RoboDK station: Config_2_New_Drillbit.rdk

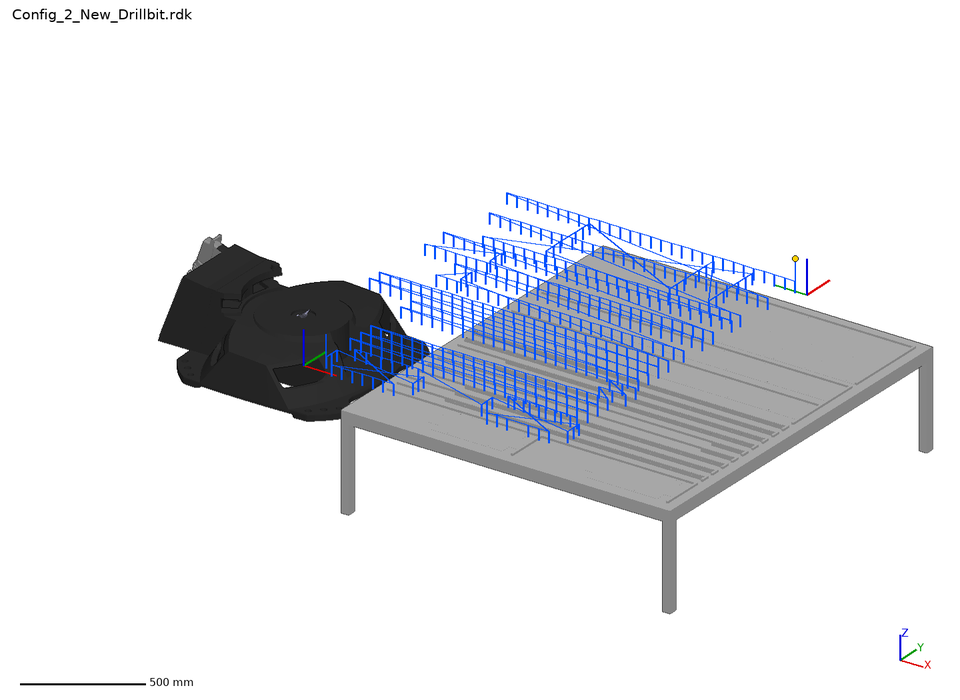
[picture v0: the station drawn from its stored meshes, robots at their saved joint values, targets as dots, program paths as lines]
Station Config_2_New_Drillbit (saved by RoboDK 5.2.3). Poses are relative to the parent item; angles as X-Y-Z fixed-axis rotations.
  - frame KUKA KR 210 R2700 extra Base at (0, 0, 0) mm
    - robot KUKA KR 210 R2700 extra: 6 axes, payload 210 kg, reach 2696 mm, repeatability 0.06 mm, weight 1068 kg
        joint limits [-185, -140, -120, -350, -125, -350] to [185, -5, 155, 350, 125, 350]; home [0, -90, 90, 0, 0, 0]; saved at [43.452, -82.309, 119.903, -52.09, 33.269, 83.396]
      - tool Spindle, TCP at (32, 0, 260) mm, rotated rx 0 ry 39 rz 0 deg, size 157.3 x 72 x 259.9 mm
  - frame Corner First Plate at (1872.67, 817.07, 510.8) mm, rotated rx 0 ry 0 rz 90 deg
  - object Table 2 at (1700, -800, 455) mm, rotated rx 0 ry 0 rz 90 deg, size 1820 x 1600 x 475 mm, geometry from Table 2.stl
  - machining project Path1 settings: rotZ(0) | rotX(0)*rotY(0) | rotz(0) | onStart | onPathStart | onApproach | onPoint | onRetract | onFinish | SetRPM(%1) | SetTool(%1) | Extruder(%1) | default | default | OutOnMov(%1) | OutOffMov(%1) | onPathFinish | M_RunCode(%1)
  - program Path1 (1332 instructions, listed below)
  - object Config_2 at (2494.97, 660, 510.8) mm, rotated rx 0 ry 0 rz 90 deg
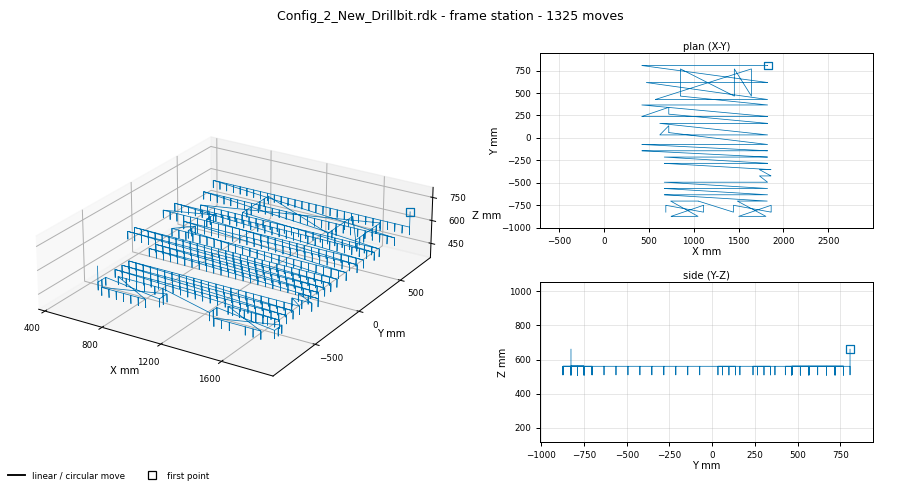
[picture p0: tool path of Config_2_New_Drillbit.rdk in frame station, 1325 of 1325 moves have a stored position in this frame; points joined in program order, loops and branches not executed]

--- program Path1 (robot KUKA KR 210 R2700 extra) ---
  Smooth(1)
  Set speed (1000.0 mm/s)
  Set Ref.: Corner First Plate
  Set Tool: Spindle
  Show Spindle
  MoveJ 1 to (-10.8, 50, 150) mm, rotated rx 180 ry 0 rz 90 deg; joints [-16.649, -45.764, 65.76, 18.984, 33.661, -29.061]
  MoveL 2 to (-10.8, 50, 150) mm, rotated rx 180 ry 0 rz 90 deg; joints [-16.649, -45.764, 65.76, 18.984, 33.661, -29.061]
  MoveL 3 to (-10.8, 50, 50) mm, rotated rx -180 ry 0 rz 90 deg; joints [-16.649, -43.606, 67.21, 20.96, 30.269, -31.389]
  MoveL 4 to (-10.8, 50, 50) mm, rotated rx -180 ry 0 rz 90 deg; joints [-16.649, -43.606, 67.21, 20.96, 30.269, -31.389]
  Set speed (150.0 mm/s)
  MoveL 5 to (-10.8, 50, -0.5) mm, rotated rx -180 ry 0 rz 90 deg; joints [-16.649, -42.409, 67.769, 22.101, 28.635, -32.7]
  MoveL 6 to (-10.8, 50, 50) mm, rotated rx -180 ry 0 rz 90 deg; joints [-16.649, -43.606, 67.21, 20.96, 30.269, -31.389]
  MoveL 7 to (-10.8, 100, 50) mm, rotated rx -180 ry 0 rz 90 deg; joints [-17.019, -45.862, 71.181, 22.479, 28.8, -33.311]
  MoveL 8 to (-10.8, 100, -0.5) mm, rotated rx 180 ry 0 rz 90 deg; joints [-17.019, -44.623, 71.727, 23.8, 27.158, -34.807]
  MoveL 9 to (-10.8, 100, 50) mm, rotated rx -180 ry 0 rz 90 deg; joints [-17.019, -45.862, 71.181, 22.479, 28.8, -33.311]
  MoveL 10 to (-10.8, 150, 50) mm, rotated rx -180 ry 0 rz 90 deg; joints [-17.405, -48.036, 74.965, 24.096, 27.458, -35.338]
  MoveL 11 to (-10.8, 150, -0.5) mm, rotated rx 180 ry 0 rz 90 deg; joints [-17.405, -46.754, 75.501, 25.621, 25.807, -37.043]
  MoveL 12 to (-10.8, 150, 50) mm, rotated rx -180 ry 0 rz 90 deg; joints [-17.405, -48.036, 74.965, 24.096, 27.458, -35.338]
  MoveL 13 to (-10.8, 200, 50) mm, rotated rx 180 ry 0 rz 90 deg; joints [-17.809, -50.14, 78.588, 25.815, 26.232, -37.474]
  MoveL 14 to (-10.8, 200, -0.5) mm, rotated rx 180 ry 0 rz 90 deg; joints [-17.809, -48.815, 79.118, 27.57, 24.574, -39.418]
  MoveL 15 to (-10.8, 200, 50) mm, rotated rx 180 ry 0 rz 90 deg; joints [-17.809, -50.14, 78.588, 25.815, 26.232, -37.474]
  MoveL 16 to (-10.8, 250, 50) mm, rotated rx -180 ry 0 rz 90 deg; joints [-18.231, -52.187, 82.07, 27.638, 25.115, -39.725]
  MoveL 17 to (-10.8, 250, -0.5) mm, rotated rx 180 ry 0 rz 90 deg; joints [-18.231, -50.817, 82.596, 29.652, 23.451, -41.935]
  MoveL 18 to (-10.8, 250, 50) mm, rotated rx -180 ry 0 rz 90 deg; joints [-18.231, -52.187, 82.07, 27.638, 25.115, -39.725]
  MoveL 19 to (-10.8, 300, 50) mm, rotated rx 180 ry 0 rz 90 deg; joints [-18.673, -54.185, 85.428, 29.564, 24.103, -42.091]
  MoveL 20 to (-10.8, 300, -0.5) mm, rotated rx 180 ry 0 rz 90 deg; joints [-18.673, -52.771, 85.952, 31.867, 22.436, -44.597]
  MoveL 21 to (-10.8, 300, 50) mm, rotated rx 180 ry 0 rz 90 deg; joints [-18.673, -54.185, 85.428, 29.564, 24.103, -42.091]
  MoveL 22 to (-10.8, 350, 50) mm, rotated rx -180 ry 0 rz 90 deg; joints [-19.137, -56.143, 88.676, 31.591, 23.192, -44.571]
  MoveL 23 to (-10.8, 350, -0.5) mm, rotated rx 180 ry 0 rz 90 deg; joints [-19.137, -54.682, 89.199, 34.212, 21.526, -47.404]
  MoveL 24 to (-10.8, 350, 50) mm, rotated rx -180 ry 0 rz 90 deg; joints [-19.137, -56.143, 88.676, 31.591, 23.192, -44.571]
  MoveL 25 to (-10.8, 400, 50) mm, rotated rx -180 ry 0 rz 90 deg; joints [-19.622, -58.067, 91.823, 33.712, 22.382, -47.16]
  MoveL 26 to (-10.8, 400, -0.5) mm, rotated rx -180 ry 0 rz 90 deg; joints [-19.622, -56.558, 92.348, 36.68, 20.72, -50.35]
  MoveL 27 to (-10.8, 400, 50) mm, rotated rx -180 ry 0 rz 90 deg; joints [-19.622, -58.067, 91.823, 33.712, 22.382, -47.16]
  MoveL 28 to (-10.8, 450, 50) mm, rotated rx -180 ry 0 rz 90 deg; joints [-20.133, -59.963, 94.88, 35.917, 21.67, -49.848]
  MoveL 29 to (-10.8, 450, -0.5) mm, rotated rx -180 ry 0 rz 90 deg; joints [-20.133, -58.405, 95.407, 39.259, 20.016, -53.424]
  MoveL 30 to (-10.8, 450, 50) mm, rotated rx -180 ry 0 rz 90 deg; joints [-20.133, -59.963, 94.88, 35.917, 21.67, -49.848]
  MoveL 31 to (-10.8, 500, 50) mm, rotated rx 180 ry 0 rz 90 deg; joints [-20.669, -61.837, 97.853, 38.19, 21.055, -52.623]
  MoveL 32 to (-10.8, 500, -0.5) mm, rotated rx -180 ry 0 rz 90 deg; joints [-20.669, -60.228, 98.385, 41.93, 19.415, -56.608]
  MoveL 33 to (-10.8, 500, 50) mm, rotated rx 180 ry 0 rz 90 deg; joints [-20.669, -61.837, 97.853, 38.19, 21.055, -52.623]
  MoveL 34 to (-10.8, 550, 50) mm, rotated rx 180 ry 0 rz 90 deg; joints [-21.233, -63.694, 100.75, 40.513, 20.539, -55.467]
  MoveL 35 to (-10.8, 550, -0.5) mm, rotated rx 180 ry 0 rz 90 deg; joints [-21.233, -62.031, 101.287, 44.668, 18.917, -59.88]
  MoveL 36 to (-10.8, 550, 50) mm, rotated rx 180 ry 0 rz 90 deg; joints [-21.233, -63.694, 100.75, 40.513, 20.539, -55.467]
  MoveL 37 to (-10.8, 600, 50) mm, rotated rx -180 ry 0 rz 90 deg; joints [-21.827, -65.538, 103.574, 42.862, 20.119, -58.358]
  MoveL 38 to (-10.8, 600, -0.5) mm, rotated rx -180 ry 0 rz 90 deg; joints [-21.827, -63.818, 104.119, 47.443, 18.521, -63.211]
  MoveL 39 to (-10.8, 600, 50) mm, rotated rx -180 ry 0 rz 90 deg; joints [-21.827, -65.538, 103.574, 42.862, 20.119, -58.358]
  MoveL 40 to (-10.8, 650, 50) mm, rotated rx 180 ry 0 rz 90 deg; joints [-22.454, -67.373, 106.332, 45.21, 19.797, -61.271]
  MoveL 41 to (-10.8, 650, -0.5) mm, rotated rx 180 ry 0 rz 90 deg; joints [-22.454, -65.594, 106.885, 50.217, 18.226, -66.566]
  MoveL 42 to (-10.8, 650, 50) mm, rotated rx 180 ry 0 rz 90 deg; joints [-22.454, -67.373, 106.332, 45.21, 19.797, -61.271]
  MoveL 43 to (-10.8, 700, 50) mm, rotated rx 180 ry 0 rz 90 deg; joints [-23.115, -69.204, 109.027, 47.525, 19.57, -64.175]
  MoveL 44 to (-10.8, 700, -0.5) mm, rotated rx 180 ry 0 rz 90 deg; joints [-23.115, -67.363, 109.589, 52.952, 18.032, -69.908]
  MoveL 45 to (-10.8, 700, 50) mm, rotated rx 180 ry 0 rz 90 deg; joints [-23.115, -69.204, 109.027, 47.525, 19.57, -64.175]
  MoveL 46 to (-10.8, 750, 50) mm, rotated rx 180 ry 0 rz 90 deg; joints [-23.815, -71.034, 111.662, 49.774, 19.44, -67.041]
  MoveL 47 to (-10.8, 750, -0.5) mm, rotated rx -180 ry 0 rz 90 deg; joints [-23.815, -69.128, 112.235, 55.606, 17.935, -73.196]
  MoveL 48 to (-10.8, 750, 50) mm, rotated rx 180 ry 0 rz 90 deg; joints [-23.815, -71.034, 111.662, 49.774, 19.44, -67.041]
  MoveL 49 to (-10.8, 800, 50) mm, rotated rx -180 ry 0 rz 90 deg; joints [-24.555, -72.868, 114.239, 51.925, 19.404, -69.836]
  MoveL 50 to (-10.8, 800, -0.5) mm, rotated rx -180 ry 0 rz 90 deg; joints [-24.555, -70.894, 114.824, 58.135, 17.935, -76.391]
  MoveL 51 to (-10.8, 800, 50) mm, rotated rx -180 ry 0 rz 90 deg; joints [-24.555, -72.868, 114.239, 51.925, 19.404, -69.836]
  MoveL 52 to (-10.8, 850, 50) mm, rotated rx 180 ry 0 rz 90 deg; joints [-25.34, -74.709, 116.761, 53.943, 19.461, -72.53]
  MoveL 53 to (-10.8, 850, -0.5) mm, rotated rx -180 ry 0 rz 90 deg; joints [-25.34, -72.663, 117.36, 60.502, 18.027, -79.455]
  MoveL 54 to (-10.8, 850, 50) mm, rotated rx 180 ry 0 rz 90 deg; joints [-25.34, -74.709, 116.761, 53.943, 19.461, -72.53]
  MoveL 55 to (-10.8, 900, 50) mm, rotated rx 180 ry 0 rz 90 deg; joints [-26.173, -76.562, 119.23, 55.799, 19.611, -75.095]
  MoveL 56 to (-10.8, 900, -0.5) mm, rotated rx 180 ry 0 rz 90 deg; joints [-26.173, -74.44, 119.843, 62.668, 18.208, -82.354]
  MoveL 57 to (-10.8, 900, 50) mm, rotated rx 180 ry 0 rz 90 deg; joints [-26.173, -76.562, 119.23, 55.799, 19.611, -75.095]
  MoveL 58 to (-10.8, 950, 50) mm, rotated rx -180 ry 0 rz 90 deg; joints [-27.059, -78.431, 121.645, 57.463, 19.851, -77.504]
  MoveL 59 to (-10.8, 950, -0.5) mm, rotated rx 180 ry 0 rz 90 deg; joints [-27.059, -76.228, 122.276, 64.603, 18.476, -85.06]
  MoveL 60 to (-10.8, 950, 50) mm, rotated rx -180 ry 0 rz 90 deg; joints [-27.059, -78.431, 121.645, 57.463, 19.851, -77.504]
  MoveL 61 to (-10.8, 1000, 50) mm, rotated rx -180 ry 0 rz 90 deg; joints [-28.001, -80.319, 124.008, 58.913, 20.182, -79.737]
  MoveL 62 to (-10.8, 1000, -0.5) mm, rotated rx -180 ry 0 rz 90 deg; joints [-28.001, -78.032, 124.658, 66.281, 18.828, -87.551]
  MoveL 63 to (-10.8, 1000, 50) mm, rotated rx -180 ry 0 rz 90 deg; joints [-28.001, -80.319, 124.008, 58.913, 20.182, -79.737]
  MoveL 64 to (-10.8, 1050, 50) mm, rotated rx 180 ry 0 rz 90 deg; joints [-29.006, -82.232, 126.32, 60.129, 20.604, -81.777]
  MoveL 65 to (-10.8, 1050, -0.5) mm, rotated rx -180 ry 0 rz 90 deg; joints [-29.006, -79.855, 126.99, 67.682, 19.261, -89.809]
  MoveL 66 to (-10.8, 1050, 50) mm, rotated rx 180 ry 0 rz 90 deg; joints [-29.006, -82.232, 126.32, 60.129, 20.604, -81.777]
  MoveL 67 to (-10.8, 1100, 50) mm, rotated rx -180 ry 0 rz 90 deg; joints [-30.078, -84.173, 128.579, 61.097, 21.117, -83.614]
  MoveL 68 to (-10.8, 1100, -0.5) mm, rotated rx -180 ry 0 rz 90 deg; joints [-30.078, -81.702, 129.272, 68.792, 19.774, -91.824]
  MoveL 69 to (-10.8, 1100, 50) mm, rotated rx -180 ry 0 rz 90 deg; joints [-30.078, -84.173, 128.579, 61.097, 21.117, -83.614]
  MoveL 70 to (-10.8, 1150, 50) mm, rotated rx -180 ry 0 rz 90 deg; joints [-31.225, -86.148, 130.786, 61.808, 21.725, -85.241]
  MoveL 71 to (-10.8, 1150, -0.5) mm, rotated rx -180 ry 0 rz 90 deg; joints [-31.225, -83.578, 131.503, 69.603, 20.369, -93.591]
  MoveL 72 to (-10.8, 1150, 50) mm, rotated rx -180 ry 0 rz 90 deg; joints [-31.225, -86.148, 130.786, 61.808, 21.725, -85.241]
  MoveL 73 to (-10.8, 1200, 50) mm, rotated rx 180 ry 0 rz 90 deg; joints [-32.452, -88.161, 132.939, 62.257, 22.43, -86.657]
  MoveL 74 to (-10.8, 1200, -0.5) mm, rotated rx -180 ry 0 rz 90 deg; joints [-32.452, -85.486, 133.682, 70.111, 21.046, -95.11]
  MoveL 75 to (-10.8, 1200, 50) mm, rotated rx 180 ry 0 rz 90 deg; joints [-32.452, -88.161, 132.939, 62.257, 22.43, -86.657]
  MoveL 76 to (-10.8, 1250, 50) mm, rotated rx -180 ry 0 rz 90 deg; joints [-33.769, -90.218, 135.035, 62.444, 23.239, -87.867]
  MoveL 77 to (-10.8, 1250, -0.5) mm, rotated rx 180 ry 0 rz 90 deg; joints [-33.769, -87.432, 135.808, 70.315, 21.809, -96.385]
  MoveL 78 to (-10.8, 1250, 50) mm, rotated rx -180 ry 0 rz 90 deg; joints [-33.769, -90.218, 135.035, 62.444, 23.239, -87.867]
  MoveL 79 to (-10.8, 1300, 50) mm, rotated rx 180 ry 0 rz 90 deg; joints [-35.182, -92.321, 137.074, 62.376, 24.158, -88.879]
  MoveL 80 to (-10.8, 1300, -0.5) mm, rotated rx -180 ry 0 rz 90 deg; joints [-35.182, -89.421, 137.879, 70.221, 22.664, -97.426]
  MoveL 81 to (-10.8, 1300, 50) mm, rotated rx 180 ry 0 rz 90 deg; joints [-35.182, -92.321, 137.074, 62.376, 24.158, -88.879]
  MoveL 82 to (-10.8, 1350, 50) mm, rotated rx -180 ry 0 rz 90 deg; joints [-36.702, -94.478, 139.052, 62.061, 25.197, -89.708]
  MoveL 83 to (-10.8, 1350, -0.5) mm, rotated rx -180 ry 0 rz 90 deg; joints [-36.702, -91.457, 139.892, 69.838, 23.62, -98.246]
  MoveL 84 to (-10.8, 1350, 50) mm, rotated rx -180 ry 0 rz 90 deg; joints [-36.702, -94.478, 139.052, 62.061, 25.197, -89.708]
  MoveL 85 to (-10.8, 1400, 50) mm, rotated rx 180 ry 0 rz 90 deg; joints [-38.338, -96.69, 140.966, 61.514, 26.368, -90.373]
  MoveL 86 to (-10.8, 1400, -0.5) mm, rotated rx 180 ry 0 rz 90 deg; joints [-38.338, -93.545, 141.843, 69.178, 24.686, -98.863]
  MoveL 87 to (-10.8, 1400, 50) mm, rotated rx 180 ry 0 rz 90 deg; joints [-38.338, -96.69, 140.966, 61.514, 26.368, -90.373]
  MoveL 88 to (-10.8, 1450, 50) mm, rotated rx 180 ry 0 rz 90 deg; joints [-40.102, -98.962, 142.811, 60.754, 27.684, -90.897]
  MoveL 89 to (-10.8, 1450, -0.5) mm, rotated rx -180 ry 0 rz 90 deg; joints [-40.102, -95.689, 143.729, 68.26, 25.875, -99.3]
  MoveL 90 to (-10.8, 1450, 50) mm, rotated rx 180 ry 0 rz 90 deg; joints [-40.102, -98.962, 142.811, 60.754, 27.684, -90.897]
  MoveL 91 to (-200, 50, 50) mm, rotated rx -180 ry 0 rz 90 deg; joints [-11.964, -45.813, 71.094, 16.522, 27.305, -24.117]
  MoveL 92 to (-200, 50, -0.5) mm, rotated rx 180 ry 0 rz 90 deg; joints [-11.964, -44.575, 71.641, 17.573, 25.599, -25.291]
  MoveL 93 to (-200, 50, 50) mm, rotated rx -180 ry 0 rz 90 deg; joints [-11.964, -45.813, 71.094, 16.522, 27.305, -24.117]
  MoveL 94 to (-200, 100, 50) mm, rotated rx 180 ry 0 rz 90 deg; joints [-12.237, -48.039, 74.969, 17.846, 25.802, -25.732]
  MoveL 95 to (-200, 100, -0.5) mm, rotated rx 180 ry 0 rz 90 deg; joints [-12.237, -46.756, 75.506, 19.085, 24.076, -27.099]
  MoveL 96 to (-200, 100, 50) mm, rotated rx 180 ry 0 rz 90 deg; joints [-12.237, -48.039, 74.969, 17.846, 25.802, -25.732]
  MoveL 97 to (-200, 150, 50) mm, rotated rx 180 ry 0 rz 90 deg; joints [-12.523, -50.194, 78.68, 19.283, 24.408, -27.465]
  MoveL 98 to (-200, 150, -0.5) mm, rotated rx -180 ry 0 rz 90 deg; joints [-12.523, -48.868, 79.21, 20.742, 22.663, -29.056]
  MoveL 99 to (-200, 150, 50) mm, rotated rx 180 ry 0 rz 90 deg; joints [-12.523, -50.194, 78.68, 19.283, 24.408, -27.465]
  MoveL 100 to (-200, 200, 50) mm, rotated rx 180 ry 0 rz 90 deg; joints [-12.823, -52.292, 82.248, 20.84, 23.117, -29.327]
  MoveL 101 to (-200, 200, -0.5) mm, rotated rx 180 ry 0 rz 90 deg; joints [-12.823, -50.92, 82.774, 22.556, 21.353, -31.181]
  MoveL 102 to (-200, 200, 50) mm, rotated rx 180 ry 0 rz 90 deg; joints [-12.823, -52.292, 82.248, 20.84, 23.117, -29.327]
  MoveL 103 to (-200, 250, 50) mm, rotated rx 180 ry 0 rz 90 deg; joints [-13.137, -54.342, 85.691, 22.527, 21.923, -31.326]
  MoveL 104 to (-200, 250, -0.5) mm, rotated rx -180 ry 0 rz 90 deg; joints [-13.137, -52.924, 86.215, 24.544, 20.142, -33.486]
  MoveL 105 to (-200, 250, 50) mm, rotated rx 180 ry 0 rz 90 deg; joints [-13.137, -54.342, 85.691, 22.527, 21.923, -31.326]
  MoveL 106 to (-200, 300, 50) mm, rotated rx -180 ry 0 rz 90 deg; joints [-13.467, -56.353, 89.022, 24.349, 20.822, -33.471]
  MoveL 107 to (-200, 300, -0.5) mm, rotated rx 180 ry 0 rz 90 deg; joints [-13.467, -54.887, 89.546, 26.715, 19.027, -35.987]
  MoveL 108 to (-200, 300, 50) mm, rotated rx -180 ry 0 rz 90 deg; joints [-13.467, -56.353, 89.022, 24.349, 20.822, -33.471]
  MoveL 109 to (-200, 350, 50) mm, rotated rx -180 ry 0 rz 90 deg; joints [-13.813, -58.332, 92.253, 26.313, 19.814, -35.768]
  MoveL 110 to (-200, 350, -0.5) mm, rotated rx 180 ry 0 rz 90 deg; joints [-13.813, -56.817, 92.779, 29.082, 18.007, -38.694]
  MoveL 111 to (-200, 350, 50) mm, rotated rx -180 ry 0 rz 90 deg; joints [-13.813, -58.332, 92.253, 26.313, 19.814, -35.768]
  MoveL 112 to (-200, 400, 50) mm, rotated rx -180 ry 0 rz 90 deg; joints [-14.177, -60.286, 95.395, 28.42, 18.897, -38.219]
  MoveL 113 to (-200, 400, -0.5) mm, rotated rx 180 ry 0 rz 90 deg; joints [-14.177, -58.719, 95.923, 31.65, 17.082, -41.615]
  MoveL 114 to (-200, 400, 50) mm, rotated rx -180 ry 0 rz 90 deg; joints [-14.177, -60.286, 95.395, 28.42, 18.897, -38.219]
  MoveL 115 to (-200, 450, 50) mm, rotated rx -180 ry 0 rz 90 deg; joints [-14.561, -62.22, 98.455, 30.667, 18.071, -40.824]
  MoveL 116 to (-200, 450, -0.5) mm, rotated rx 180 ry 0 rz 90 deg; joints [-14.561, -60.6, 98.987, 34.419, 16.255, -44.75]
  MoveL 117 to (-200, 450, 50) mm, rotated rx -180 ry 0 rz 90 deg; joints [-14.561, -62.22, 98.455, 30.667, 18.071, -40.824]
  MoveL 118 to (-200, 500, 50) mm, rotated rx 180 ry 0 rz 90 deg; joints [-14.965, -64.141, 101.439, 33.046, 17.338, -43.575]
  MoveL 119 to (-200, 500, -0.5) mm, rotated rx 180 ry 0 rz 90 deg; joints [-14.965, -62.464, 101.978, 37.38, 15.527, -48.093]
  MoveL 120 to (-200, 500, 50) mm, rotated rx 180 ry 0 rz 90 deg; joints [-14.965, -64.141, 101.439, 33.046, 17.338, -43.575]
  MoveL 121 to (-200, 550, 50) mm, rotated rx -180 ry 0 rz 90 deg; joints [-15.392, -66.053, 104.355, 35.542, 16.699, -46.459]
  MoveL 122 to (-200, 550, -0.5) mm, rotated rx 180 ry 0 rz 90 deg; joints [-15.392, -64.317, 104.901, 40.513, 14.9, -51.624]
  MoveL 123 to (-200, 550, 50) mm, rotated rx -180 ry 0 rz 90 deg; joints [-15.392, -66.053, 104.355, 35.542, 16.699, -46.459]
  MoveL 124 to (-200, 600, 50) mm, rotated rx 180 ry 0 rz 90 deg; joints [-15.843, -67.962, 107.206, 38.131, 16.156, -49.453]
  MoveL 125 to (-200, 600, -0.5) mm, rotated rx 180 ry 0 rz 90 deg; joints [-15.843, -66.164, 107.761, 43.787, 14.376, -55.314]
  MoveL 126 to (-200, 600, 50) mm, rotated rx 180 ry 0 rz 90 deg; joints [-15.843, -67.962, 107.206, 38.131, 16.156, -49.453]
  MoveL 127 to (-200, 650, 50) mm, rotated rx -180 ry 0 rz 90 deg; joints [-16.321, -69.873, 109.997, 40.781, 15.71, -52.526]
  MoveL 128 to (-200, 650, -0.5) mm, rotated rx -180 ry 0 rz 90 deg; joints [-16.321, -68.009, 110.563, 47.155, 13.958, -59.118]
  MoveL 129 to (-200, 650, 50) mm, rotated rx -180 ry 0 rz 90 deg; joints [-16.321, -69.873, 109.997, 40.781, 15.71, -52.526]
  MoveL 130 to (-200, 700, 50) mm, rotated rx -180 ry 0 rz 90 deg; joints [-16.828, -71.79, 112.732, 43.453, 15.361, -55.64]
  MoveL 131 to (-200, 700, -0.5) mm, rotated rx -180 ry 0 rz 90 deg; joints [-16.828, -69.857, 113.31, 50.559, 13.645, -62.979]
  MoveL 132 to (-200, 700, 50) mm, rotated rx -180 ry 0 rz 90 deg; joints [-16.828, -71.79, 112.732, 43.453, 15.361, -55.64]
  MoveL 133 to (-200, 750, 50) mm, rotated rx 180 ry 0 rz 90 deg; joints [-17.366, -73.72, 115.414, 46.097, 15.112, -58.749]
  MoveL 134 to (-200, 750, -0.5) mm, rotated rx -180 ry 0 rz 90 deg; joints [-17.366, -71.713, 116.005, 53.929, 13.438, -66.829]
  MoveL 135 to (-200, 750, 50) mm, rotated rx 180 ry 0 rz 90 deg; joints [-17.366, -73.72, 115.414, 46.097, 15.112, -58.749]
  MoveL 136 to (-200, 800, 50) mm, rotated rx 180 ry 0 rz 90 deg; joints [-17.939, -75.667, 118.045, 48.66, 14.961, -61.8]
  MoveL 137 to (-200, 800, -0.5) mm, rotated rx -180 ry 0 rz 90 deg; joints [-17.939, -73.581, 118.652, 57.189, 13.334, -70.594]
  MoveL 138 to (-200, 800, 50) mm, rotated rx 180 ry 0 rz 90 deg; joints [-17.939, -75.667, 118.045, 48.66, 14.961, -61.8]
  MoveL 139 to (-200, 850, 50) mm, rotated rx -180 ry 0 rz 90 deg; joints [-18.549, -77.637, 120.627, 51.085, 14.91, -64.738]
  MoveL 140 to (-200, 850, -0.5) mm, rotated rx 180 ry 0 rz 90 deg; joints [-18.549, -75.469, 121.251, 60.261, 13.33, -74.198]
  MoveL 141 to (-200, 850, 50) mm, rotated rx -180 ry 0 rz 90 deg; joints [-18.549, -77.637, 120.627, 51.085, 14.91, -64.738]
  MoveL 142 to (-200, 900, 50) mm, rotated rx 180 ry 0 rz 90 deg; joints [-19.2, -79.636, 123.163, 53.316, 14.956, -67.509]
  MoveL 143 to (-200, 900, -0.5) mm, rotated rx -180 ry 0 rz 90 deg; joints [-19.2, -77.38, 123.805, 63.074, 13.423, -77.572]
  MoveL 144 to (-200, 900, 50) mm, rotated rx 180 ry 0 rz 90 deg; joints [-19.2, -79.636, 123.163, 53.316, 14.956, -67.509]
  MoveL 145 to (-200, 950, 50) mm, rotated rx 180 ry 0 rz 90 deg; joints [-19.898, -81.672, 125.652, 55.3, 15.101, -70.063]
  MoveL 146 to (-200, 950, -0.5) mm, rotated rx -180 ry 0 rz 90 deg; joints [-19.898, -79.322, 126.316, 65.561, 13.607, -80.651]
  MoveL 147 to (-200, 950, 50) mm, rotated rx 180 ry 0 rz 90 deg; joints [-19.898, -81.672, 125.652, 55.3, 15.101, -70.063]
  MoveL 148 to (-200, 1000, 50) mm, rotated rx 180 ry 0 rz 90 deg; joints [-20.645, -83.751, 128.096, 56.99, 15.343, -72.353]
  MoveL 149 to (-200, 1000, -0.5) mm, rotated rx -180 ry 0 rz 90 deg; joints [-20.645, -81.301, 128.783, 67.668, 13.879, -83.385]
  MoveL 150 to (-200, 1000, 50) mm, rotated rx 180 ry 0 rz 90 deg; joints [-20.645, -83.751, 128.096, 56.99, 15.343, -72.353]
  MoveL 151 to (-200, 1050, 50) mm, rotated rx -180 ry 0 rz 90 deg; joints [-21.448, -85.883, 130.495, 58.346, 15.684, -74.344]
  MoveL 152 to (-200, 1050, -0.5) mm, rotated rx 180 ry 0 rz 90 deg; joints [-21.448, -83.326, 131.208, 69.353, 14.235, -85.735]
  MoveL 153 to (-200, 1050, 50) mm, rotated rx -180 ry 0 rz 90 deg; joints [-21.448, -85.883, 130.495, 58.346, 15.684, -74.344]
  MoveL 154 to (-200, 1100, 50) mm, rotated rx 180 ry 0 rz 90 deg; joints [-22.312, -88.075, 132.849, 59.338, 16.126, -76.008]
  MoveL 155 to (-200, 1100, -0.5) mm, rotated rx -180 ry 0 rz 90 deg; joints [-22.312, -85.405, 133.591, 70.587, 14.674, -87.672]
  MoveL 156 to (-200, 1100, 50) mm, rotated rx 180 ry 0 rz 90 deg; joints [-22.312, -88.075, 132.849, 59.338, 16.126, -76.008]
  MoveL 157 to (-200, 1150, 50) mm, rotated rx 180 ry 0 rz 90 deg; joints [-23.246, -90.339, 135.156, 59.946, 16.676, -77.327]
  MoveL 158 to (-200, 1150, -0.5) mm, rotated rx -180 ry 0 rz 90 deg; joints [-23.246, -87.547, 135.931, 71.348, 15.197, -89.182]
  MoveL 159 to (-200, 1150, 50) mm, rotated rx 180 ry 0 rz 90 deg; joints [-23.246, -90.339, 135.156, 59.946, 16.676, -77.327]
  MoveL 160 to (-200, 1200, 50) mm, rotated rx -180 ry 0 rz 90 deg; joints [-24.255, -92.686, 137.417, 60.159, 17.34, -78.294]
  MoveL 161 to (-200, 1200, -0.5) mm, rotated rx -180 ry 0 rz 90 deg; joints [-24.255, -89.766, 138.228, 71.627, 15.808, -90.255]
  MoveL 162 to (-200, 1200, 50) mm, rotated rx -180 ry 0 rz 90 deg; joints [-24.255, -92.686, 137.417, 60.159, 17.34, -78.294]
  MoveL 163 to (-200, 1250, 50) mm, rotated rx -180 ry 0 rz 90 deg; joints [-25.351, -95.13, 139.628, 59.978, 18.132, -78.912]
  MoveL 164 to (-200, 1250, -0.5) mm, rotated rx 180 ry 0 rz 90 deg; joints [-25.351, -92.072, 140.479, 71.421, 16.515, -90.893]
  MoveL 165 to (-200, 1250, 50) mm, rotated rx -180 ry 0 rz 90 deg; joints [-25.351, -95.13, 139.628, 59.978, 18.132, -78.912]
  MoveL 166 to (-200, 1300, 50) mm, rotated rx 180 ry 0 rz 90 deg; joints [-26.542, -97.684, 141.787, 59.412, 19.067, -79.192]
  MoveL 167 to (-200, 1300, -0.5) mm, rotated rx -180 ry 0 rz 90 deg; joints [-26.542, -94.482, 142.682, 70.734, 17.332, -91.105]
  MoveL 168 to (-200, 1300, 50) mm, rotated rx 180 ry 0 rz 90 deg; joints [-26.542, -97.684, 141.787, 59.412, 19.067, -79.192]
  MoveL 169 to (-200, 1350, 50) mm, rotated rx 180 ry 0 rz 90 deg; joints [-27.842, -100.365, 143.891, 58.481, 20.169, -79.16]
  MoveL 170 to (-200, 1350, -0.5) mm, rotated rx -180 ry 0 rz 90 deg; joints [-27.842, -97.013, 144.835, 69.582, 18.278, -90.91]
  MoveL 171 to (-200, 1350, 50) mm, rotated rx 180 ry 0 rz 90 deg; joints [-27.842, -100.365, 143.891, 58.481, 20.169, -79.16]
  MoveL 172 to (-200, 1400, 50) mm, rotated rx 180 ry 0 rz 90 deg; joints [-29.264, -103.192, 145.935, 57.218, 21.464, -78.849]
  MoveL 173 to (-200, 1400, -0.5) mm, rotated rx 180 ry 0 rz 90 deg; joints [-29.264, -99.683, 146.934, 67.989, 19.379, -90.335]
  MoveL 174 to (-200, 1400, 50) mm, rotated rx 180 ry 0 rz 90 deg; joints [-29.264, -103.192, 145.935, 57.218, 21.464, -78.849]
  MoveL 175 to (-389.2, 50, 50) mm, rotated rx 180 ry 0 rz 90 deg; joints [-7.11, -47.25, 73.601, 10.527, 25.238, -15.078]
  MoveL 176 to (-389.2, 50, -0.5) mm, rotated rx 180 ry 0 rz 90 deg; joints [-7.11, -45.983, 74.141, 11.282, 23.464, -15.907]
  MoveL 177 to (-389.2, 50, 50) mm, rotated rx 180 ry 0 rz 90 deg; joints [-7.11, -47.25, 73.601, 10.527, 25.238, -15.078]
  MoveL 178 to (-389.2, 100, 50) mm, rotated rx -180 ry 0 rz 90 deg; joints [-7.276, -49.462, 77.424, 11.445, 23.684, -16.17]
  MoveL 179 to (-389.2, 100, -0.5) mm, rotated rx 180 ry 0 rz 90 deg; joints [-7.276, -48.151, 77.957, 12.35, 21.88, -17.151]
  MoveL 180 to (-389.2, 100, 50) mm, rotated rx -180 ry 0 rz 90 deg; joints [-7.276, -49.462, 77.424, 11.445, 23.684, -16.17]
  MoveL 181 to (-389.2, 150, 50) mm, rotated rx -180 ry 0 rz 90 deg; joints [-7.45, -51.612, 81.096, 12.457, 22.227, -17.36]
  MoveL 182 to (-389.2, 150, -0.5) mm, rotated rx 180 ry 0 rz 90 deg; joints [-7.45, -50.255, 81.624, 13.544, 20.391, -18.526]
  MoveL 183 to (-389.2, 150, 50) mm, rotated rx -180 ry 0 rz 90 deg; joints [-7.45, -51.612, 81.096, 12.457, 22.227, -17.36]
  MoveL 184 to (-389.2, 200, 50) mm, rotated rx 180 ry 0 rz 90 deg; joints [-7.632, -53.711, 84.636, 13.576, 20.859, -18.661]
  MoveL 185 to (-389.2, 200, -0.5) mm, rotated rx 180 ry 0 rz 90 deg; joints [-7.632, -52.308, 85.161, 14.884, 18.99, -20.052]
  MoveL 186 to (-389.2, 200, 50) mm, rotated rx 180 ry 0 rz 90 deg; joints [-7.632, -53.711, 84.636, 13.576, 20.859, -18.661]
  MoveL 187 to (-389.2, 250, 50) mm, rotated rx 180 ry 0 rz 90 deg; joints [-7.823, -55.769, 88.06, 14.814, 19.575, -20.087]
  MoveL 188 to (-389.2, 250, -0.5) mm, rotated rx 180 ry 0 rz 90 deg; joints [-7.823, -54.318, 88.583, 16.391, 17.672, -21.751]
  MoveL 189 to (-389.2, 250, 50) mm, rotated rx 180 ry 0 rz 90 deg; joints [-7.823, -55.769, 88.06, 14.814, 19.575, -20.087]
  MoveL 190 to (-389.2, 300, 50) mm, rotated rx 180 ry 0 rz 90 deg; joints [-8.024, -57.794, 91.38, 16.184, 18.372, -21.652]
  MoveL 191 to (-389.2, 300, -0.5) mm, rotated rx 180 ry 0 rz 90 deg; joints [-8.024, -56.292, 91.904, 18.089, 16.435, -23.648]
  MoveL 192 to (-389.2, 300, 50) mm, rotated rx 180 ry 0 rz 90 deg; joints [-8.024, -57.794, 91.38, 16.184, 18.372, -21.652]
  MoveL 193 to (-389.2, 350, 50) mm, rotated rx -180 ry 0 rz 90 deg; joints [-8.236, -59.793, 94.607, 17.701, 17.247, -23.37]
  MoveL 194 to (-389.2, 350, -0.5) mm, rotated rx 180 ry 0 rz 90 deg; joints [-8.236, -58.239, 95.134, 20.006, 15.278, -25.771]
  MoveL 195 to (-389.2, 350, 50) mm, rotated rx -180 ry 0 rz 90 deg; joints [-8.236, -59.793, 94.607, 17.701, 17.247, -23.37]
  MoveL 196 to (-389.2, 400, 50) mm, rotated rx 180 ry 0 rz 90 deg; joints [-8.459, -61.772, 97.75, 19.377, 16.201, -25.254]
  MoveL 197 to (-389.2, 400, -0.5) mm, rotated rx 180 ry 0 rz 90 deg; joints [-8.459, -60.164, 98.281, 22.17, 14.2, -28.149]
  MoveL 198 to (-389.2, 400, 50) mm, rotated rx 180 ry 0 rz 90 deg; joints [-8.459, -61.772, 97.75, 19.377, 16.201, -25.254]
  MoveL 199 to (-389.2, 450, 50) mm, rotated rx 180 ry 0 rz 90 deg; joints [-8.694, -63.738, 100.817, 21.225, 15.234, -27.319]
  MoveL 200 to (-389.2, 450, -0.5) mm, rotated rx -180 ry 0 rz 90 deg; joints [-8.694, -62.073, 101.354, 24.61, 13.205, -30.811]
  MoveL 201 to (-389.2, 450, 50) mm, rotated rx 180 ry 0 rz 90 deg; joints [-8.694, -63.738, 100.817, 21.225, 15.234, -27.319]
  MoveL 202 to (-389.2, 500, 50) mm, rotated rx 180 ry 0 rz 90 deg; joints [-8.943, -65.696, 103.815, 23.253, 14.347, -29.574]
  MoveL 203 to (-389.2, 500, -0.5) mm, rotated rx 180 ry 0 rz 90 deg; joints [-8.943, -63.972, 104.359, 27.352, 12.293, -33.785]
  MoveL 204 to (-389.2, 500, 50) mm, rotated rx 180 ry 0 rz 90 deg; joints [-8.943, -65.696, 103.815, 23.253, 14.347, -29.574]
  MoveL 205 to (-389.2, 550, 50) mm, rotated rx 180 ry 0 rz 90 deg; joints [-9.206, -67.653, 106.748, 25.466, 13.541, -32.023]
  MoveL 206 to (-389.2, 550, -0.5) mm, rotated rx -180 ry 0 rz 90 deg; joints [-9.206, -65.865, 107.302, 30.415, 11.471, -37.092]
  MoveL 207 to (-389.2, 550, 50) mm, rotated rx 180 ry 0 rz 90 deg; joints [-9.206, -67.653, 106.748, 25.466, 13.541, -32.023]
  MoveL 208 to (-389.2, 600, 50) mm, rotated rx 180 ry 0 rz 90 deg; joints [-9.485, -69.614, 109.623, 27.86, 12.821, -34.664]
  MoveL 209 to (-389.2, 600, -0.5) mm, rotated rx -180 ry 0 rz 90 deg; joints [-9.485, -67.759, 110.187, 33.808, 10.741, -40.739]
  MoveL 210 to (-389.2, 600, 50) mm, rotated rx 180 ry 0 rz 90 deg; joints [-9.485, -69.614, 109.623, 27.86, 12.821, -34.664]
  MoveL 211 to (-389.2, 650, 50) mm, rotated rx 180 ry 0 rz 90 deg; joints [-9.781, -71.584, 112.442, 30.419, 12.19, -37.482]
  MoveL 212 to (-389.2, 650, -0.5) mm, rotated rx 180 ry 0 rz 90 deg; joints [-9.781, -69.658, 113.018, 37.518, 10.11, -44.716]
  MoveL 213 to (-389.2, 650, 50) mm, rotated rx 180 ry 0 rz 90 deg; joints [-9.781, -71.584, 112.442, 30.419, 12.19, -37.482]
  MoveL 214 to (-389.2, 700, 50) mm, rotated rx 180 ry 0 rz 90 deg; joints [-10.096, -73.571, 115.21, 33.115, 11.65, -40.45]
  MoveL 215 to (-389.2, 700, -0.5) mm, rotated rx -180 ry 0 rz 90 deg; joints [-10.096, -71.569, 115.8, 41.503, 9.583, -48.982]
  MoveL 216 to (-389.2, 700, 50) mm, rotated rx 180 ry 0 rz 90 deg; joints [-10.096, -73.571, 115.21, 33.115, 11.65, -40.45]
  MoveL 217 to (-389.2, 750, 50) mm, rotated rx 180 ry 0 rz 90 deg; joints [-10.432, -75.579, 117.929, 35.9, 11.205, -43.52]
  MoveL 218 to (-389.2, 750, -0.5) mm, rotated rx 180 ry 0 rz 90 deg; joints [-10.432, -73.498, 118.535, 45.687, 9.163, -53.461]
  MoveL 219 to (-389.2, 750, 50) mm, rotated rx 180 ry 0 rz 90 deg; joints [-10.432, -75.579, 117.929, 35.9, 11.205, -43.52]
  MoveL 220 to (-389.2, 800, 50) mm, rotated rx 180 ry 0 rz 90 deg; joints [-10.79, -77.617, 120.603, 38.709, 10.859, -46.629]
  MoveL 221 to (-389.2, 800, -0.5) mm, rotated rx -180 ry 0 rz 90 deg; joints [-10.79, -75.45, 121.226, 49.953, 8.853, -58.039]
  MoveL 222 to (-389.2, 800, 50) mm, rotated rx 180 ry 0 rz 90 deg; joints [-10.79, -77.617, 120.603, 38.709, 10.859, -46.629]
  MoveL 223 to (-389.2, 850, 50) mm, rotated rx -180 ry 0 rz 90 deg; joints [-11.174, -79.692, 123.233, 41.458, 10.615, -49.696]
  MoveL 224 to (-389.2, 850, -0.5) mm, rotated rx 180 ry 0 rz 90 deg; joints [-11.174, -77.434, 123.876, 54.153, 8.653, -62.568]
  MoveL 225 to (-389.2, 850, 50) mm, rotated rx -180 ry 0 rz 90 deg; joints [-11.174, -79.692, 123.233, 41.458, 10.615, -49.696]
  MoveL 226 to (-389.2, 900, 50) mm, rotated rx 180 ry 0 rz 90 deg; joints [-11.586, -81.813, 125.82, 44.052, 10.473, -52.623]
  MoveL 227 to (-389.2, 900, -0.5) mm, rotated rx -180 ry 0 rz 90 deg; joints [-11.586, -79.456, 126.486, 58.117, 8.56, -66.881]
  MoveL 228 to (-389.2, 900, 50) mm, rotated rx 180 ry 0 rz 90 deg; joints [-11.586, -81.813, 125.82, 44.052, 10.473, -52.623]
  MoveL 229 to (-389.2, 950, 50) mm, rotated rx -180 ry 0 rz 90 deg; joints [-12.028, -83.988, 128.368, 46.385, 10.437, -55.31]
  MoveL 230 to (-389.2, 950, -0.5) mm, rotated rx 180 ry 0 rz 90 deg; joints [-12.028, -81.526, 129.058, 61.675, 8.568, -70.808]
  MoveL 231 to (-389.2, 950, 50) mm, rotated rx -180 ry 0 rz 90 deg; joints [-12.028, -83.988, 128.368, 46.385, 10.437, -55.31]
  MoveL 232 to (-389.2, 1000, 50) mm, rotated rx -180 ry 0 rz 90 deg; joints [-12.506, -86.229, 130.875, 48.356, 10.507, -57.654]
  MoveL 233 to (-389.2, 1000, -0.5) mm, rotated rx 180 ry 0 rz 90 deg; joints [-12.506, -83.655, 131.593, 64.671, 8.671, -74.195]
  MoveL 234 to (-389.2, 1000, 50) mm, rotated rx -180 ry 0 rz 90 deg; joints [-12.506, -86.229, 130.875, 48.356, 10.507, -57.654]
  MoveL 235 to (-389.2, 1050, 50) mm, rotated rx 180 ry 0 rz 90 deg; joints [-13.022, -88.55, 133.342, 49.872, 10.688, -59.566]
  MoveL 236 to (-389.2, 1050, -0.5) mm, rotated rx -180 ry 0 rz 90 deg; joints [-13.022, -85.854, 134.092, 66.976, 8.863, -76.916]
  MoveL 237 to (-389.2, 1050, 50) mm, rotated rx 180 ry 0 rz 90 deg; joints [-13.022, -88.55, 133.342, 49.872, 10.688, -59.566]
  MoveL 238 to (-389.2, 1100, 50) mm, rotated rx -180 ry 0 rz 90 deg; joints [-13.582, -90.963, 135.77, 50.859, 10.985, -60.973]
  MoveL 239 to (-389.2, 1100, -0.5) mm, rotated rx -180 ry 0 rz 90 deg; joints [-13.582, -88.137, 136.554, 68.496, 9.14, -78.879]
  MoveL 240 to (-389.2, 1100, 50) mm, rotated rx -180 ry 0 rz 90 deg; joints [-13.582, -90.963, 135.77, 50.859, 10.985, -60.973]
  MoveL 241 to (-389.2, 1150, 50) mm, rotated rx -180 ry 0 rz 90 deg; joints [-14.191, -93.488, 138.158, 51.266, 11.407, -61.825]
  MoveL 242 to (-389.2, 1150, -0.5) mm, rotated rx 180 ry 0 rz 90 deg; joints [-14.191, -90.522, 138.981, 69.168, 9.501, -80.021]
  MoveL 243 to (-389.2, 1150, 50) mm, rotated rx -180 ry 0 rz 90 deg; joints [-14.191, -93.488, 138.158, 51.266, 11.407, -61.825]
  MoveL 244 to (-389.2, 1200, 50) mm, rotated rx 180 ry 0 rz 90 deg; joints [-14.856, -96.143, 140.504, 51.069, 11.971, -62.1]
  MoveL 245 to (-389.2, 1200, -0.5) mm, rotated rx 180 ry 0 rz 90 deg; joints [-14.856, -93.029, 141.371, 68.956, 9.955, -80.31]
  MoveL 246 to (-389.2, 1200, 50) mm, rotated rx 180 ry 0 rz 90 deg; joints [-14.856, -96.143, 140.504, 51.069, 11.971, -62.1]
  MoveL 247 to (-389.2, 1250, 50) mm, rotated rx 180 ry 0 rz 90 deg; joints [-15.585, -98.955, 142.806, 50.275, 12.699, -61.806]
  MoveL 248 to (-389.2, 1250, -0.5) mm, rotated rx 180 ry 0 rz 90 deg; joints [-15.585, -95.682, 143.723, 67.852, 10.518, -79.741]
  MoveL 249 to (-389.2, 1250, 50) mm, rotated rx 180 ry 0 rz 90 deg; joints [-15.585, -98.955, 142.806, 50.275, 12.699, -61.806]
  MoveL 250 to (-389.2, 1300, 50) mm, rotated rx 180 ry 0 rz 90 deg; joints [-16.386, -101.952, 145.06, 48.919, 13.623, -60.98]
  MoveL 251 to (-389.2, 1300, -0.5) mm, rotated rx 180 ry 0 rz 90 deg; joints [-16.386, -98.511, 146.035, 65.88, 11.217, -78.337]
  MoveL 252 to (-389.2, 1300, 50) mm, rotated rx 180 ry 0 rz 90 deg; joints [-16.386, -101.952, 145.06, 48.919, 13.623, -60.98]
  MoveL 253 to (-48.6, 230, 50) mm, rotated rx 180 ry 0 rz 90 deg; joints [-17.072, -51.863, 81.522, 26.069, 24.86, -37.359]
  MoveL 254 to (-48.6, 230, -0.5) mm, rotated rx 180 ry 0 rz 90 deg; joints [-17.072, -50.501, 82.048, 27.995, 23.178, -39.468]
  MoveL 255 to (-48.6, 230, 50) mm, rotated rx 180 ry 0 rz 90 deg; joints [-17.072, -51.863, 81.522, 26.069, 24.86, -37.359]
  MoveL 256 to (-98.6, 230, 50) mm, rotated rx 180 ry 0 rz 90 deg; joints [-15.747, -52.464, 82.539, 24.838, 23.991, -35.283]
  MoveL 257 to (-98.6, 230, -0.5) mm, rotated rx -180 ry 0 rz 90 deg; joints [-15.747, -51.089, 83.065, 26.776, 22.28, -37.39]
  MoveL 258 to (-98.6, 230, 50) mm, rotated rx 180 ry 0 rz 90 deg; joints [-15.747, -52.464, 82.539, 24.838, 23.991, -35.283]
  MoveL 259 to (-148.6, 230, 50) mm, rotated rx 180 ry 0 rz 90 deg; joints [-14.406, -53.014, 83.466, 23.446, 23.173, -33.026]
  MoveL 260 to (-148.6, 230, -0.5) mm, rotated rx -180 ry 0 rz 90 deg; joints [-14.406, -51.627, 83.991, 25.373, 21.431, -35.109]
  MoveL 261 to (-148.6, 230, 50) mm, rotated rx 180 ry 0 rz 90 deg; joints [-14.406, -53.014, 83.466, 23.446, 23.173, -33.026]
  MoveL 262 to (-251.4, 230, 50) mm, rotated rx -180 ry 0 rz 90 deg; joints [-11.598, -53.986, 85.096, 20.04, 21.667, -27.788]
  MoveL 263 to (-251.4, 230, -0.5) mm, rotated rx 180 ry 0 rz 90 deg; joints [-11.598, -52.576, 85.62, 21.864, 19.861, -29.739]
  MoveL 264 to (-251.4, 230, 50) mm, rotated rx -180 ry 0 rz 90 deg; joints [-11.598, -53.986, 85.096, 20.04, 21.667, -27.788]
  MoveL 265 to (-301.4, 230, 50) mm, rotated rx 180 ry 0 rz 90 deg; joints [-10.211, -54.381, 85.755, 18.112, 21.029, -24.946]
  MoveL 266 to (-301.4, 230, -0.5) mm, rotated rx 180 ry 0 rz 90 deg; joints [-10.211, -52.962, 86.279, 19.838, 19.192, -26.783]
  MoveL 267 to (-301.4, 230, 50) mm, rotated rx 180 ry 0 rz 90 deg; joints [-10.211, -54.381, 85.755, 18.112, 21.029, -24.946]
  MoveL 268 to (-351.4, 230, 50) mm, rotated rx -180 ry 0 rz 90 deg; joints [-8.811, -54.725, 86.328, 16.008, 20.46, -21.914]
  MoveL 269 to (-351.4, 230, -0.5) mm, rotated rx 180 ry 0 rz 90 deg; joints [-8.811, -53.298, 86.852, 17.598, 18.593, -23.601]
  MoveL 270 to (-351.4, 230, 50) mm, rotated rx -180 ry 0 rz 90 deg; joints [-8.811, -54.725, 86.328, 16.008, 20.46, -21.914]
  MoveL 271 to (-48.6, 420, 50) mm, rotated rx 180 ry 0 rz 90 deg; joints [-18.752, -59.332, 93.867, 33.787, 21.334, -46.713]
  MoveL 272 to (-48.6, 420, -0.5) mm, rotated rx -180 ry 0 rz 90 deg; joints [-18.752, -57.791, 94.394, 36.992, 19.647, -50.135]
  MoveL 273 to (-48.6, 420, 50) mm, rotated rx 180 ry 0 rz 90 deg; joints [-18.752, -59.332, 93.867, 33.787, 21.334, -46.713]
  MoveL 274 to (-98.6, 420, 50) mm, rotated rx -180 ry 0 rz 90 deg; joints [-17.314, -59.954, 94.865, 32.547, 20.373, -44.511]
  MoveL 275 to (-98.6, 420, -0.5) mm, rotated rx -180 ry 0 rz 90 deg; joints [-17.314, -58.396, 95.393, 35.857, 18.647, -48.021]
  MoveL 276 to (-98.6, 420, 50) mm, rotated rx -180 ry 0 rz 90 deg; joints [-17.314, -59.954, 94.865, 32.547, 20.373, -44.511]
  MoveL 277 to (-148.6, 420, 50) mm, rotated rx 180 ry 0 rz 90 deg; joints [-15.853, -60.526, 95.778, 31.078, 19.453, -42.055]
  MoveL 278 to (-148.6, 420, -0.5) mm, rotated rx 180 ry 0 rz 90 deg; joints [-15.853, -58.953, 96.307, 34.466, 17.684, -45.628]
  MoveL 279 to (-148.6, 420, 50) mm, rotated rx 180 ry 0 rz 90 deg; joints [-15.853, -60.526, 95.778, 31.078, 19.453, -42.055]
  MoveL 280 to (-251.4, 420, 50) mm, rotated rx 180 ry 0 rz 90 deg; joints [-12.783, -61.543, 97.389, 27.234, 17.715, -36.117]
  MoveL 281 to (-251.4, 420, -0.5) mm, rotated rx 180 ry 0 rz 90 deg; joints [-12.783, -59.941, 97.92, 30.657, 15.848, -39.692]
  MoveL 282 to (-251.4, 420, 50) mm, rotated rx 180 ry 0 rz 90 deg; joints [-12.783, -61.543, 97.389, 27.234, 17.715, -36.117]
  MoveL 283 to (-301.4, 420, 50) mm, rotated rx 180 ry 0 rz 90 deg; joints [-11.262, -61.958, 98.043, 24.919, 16.959, -32.757]
  MoveL 284 to (-301.4, 420, -0.5) mm, rotated rx 180 ry 0 rz 90 deg; joints [-11.262, -60.345, 98.575, 28.27, 15.04, -36.241]
  MoveL 285 to (-301.4, 420, 50) mm, rotated rx 180 ry 0 rz 90 deg; joints [-11.262, -61.958, 98.043, 24.919, 16.959, -32.757]
  MoveL 286 to (-351.4, 420, 50) mm, rotated rx 180 ry 0 rz 90 deg; joints [-9.724, -62.321, 98.612, 22.292, 16.272, -29.068]
  MoveL 287 to (-351.4, 420, -0.5) mm, rotated rx -180 ry 0 rz 90 deg; joints [-9.724, -60.697, 99.145, 25.489, 14.3, -32.381]
  MoveL 288 to (-351.4, 420, 50) mm, rotated rx 180 ry 0 rz 90 deg; joints [-9.724, -62.321, 98.612, 22.292, 16.272, -29.068]
  MoveL 289 to (-48.6, 1020, 50) mm, rotated rx -180 ry 0 rz 90 deg; joints [-26.981, -81.847, 125.862, 59.347, 19.384, -79.447]
  MoveL 290 to (-48.6, 1020, -0.5) mm, rotated rx 180 ry 0 rz 90 deg; joints [-26.981, -79.489, 126.528, 67.339, 18.024, -87.882]
  MoveL 291 to (-48.6, 1020, 50) mm, rotated rx -180 ry 0 rz 90 deg; joints [-26.981, -81.847, 125.862, 59.347, 19.384, -79.447]
  MoveL 292 to (-98.6, 1020, 50) mm, rotated rx -180 ry 0 rz 90 deg; joints [-25.055, -82.815, 127.008, 59.052, 18.105, -77.72]
  MoveL 293 to (-98.6, 1020, -0.5) mm, rotated rx 180 ry 0 rz 90 deg; joints [-25.055, -80.41, 127.684, 67.851, 16.723, -86.939]
  MoveL 294 to (-98.6, 1020, 50) mm, rotated rx -180 ry 0 rz 90 deg; joints [-25.055, -82.815, 127.008, 59.052, 18.105, -77.72]
  MoveL 295 to (-148.6, 1020, 50) mm, rotated rx 180 ry 0 rz 90 deg; joints [-23.066, -83.726, 128.066, 58.494, 16.81, -75.68]
  MoveL 296 to (-148.6, 1020, -0.5) mm, rotated rx 180 ry 0 rz 90 deg; joints [-23.066, -81.277, 128.753, 68.217, 15.398, -85.797]
  MoveL 297 to (-148.6, 1020, 50) mm, rotated rx 180 ry 0 rz 90 deg; joints [-23.066, -83.726, 128.066, 58.494, 16.81, -75.68]
  MoveL 298 to (-251.4, 1020, 50) mm, rotated rx 180 ry 0 rz 90 deg; joints [-18.79, -85.398, 129.958, 56.203, 14.119, -70.197]
  MoveL 299 to (-251.4, 1020, -0.5) mm, rotated rx -180 ry 0 rz 90 deg; joints [-18.79, -82.865, 130.666, 68.302, 12.601, -82.629]
  MoveL 300 to (-251.4, 1020, 50) mm, rotated rx 180 ry 0 rz 90 deg; joints [-18.79, -85.398, 129.958, 56.203, 14.119, -70.197]
  MoveL 301 to (-301.4, 1020, 50) mm, rotated rx -180 ry 0 rz 90 deg; joints [-16.626, -86.102, 130.736, 54.303, 12.81, -66.681]
  MoveL 302 to (-301.4, 1020, -0.5) mm, rotated rx -180 ry 0 rz 90 deg; joints [-16.626, -83.534, 131.452, 67.852, 11.21, -80.529]
  MoveL 303 to (-301.4, 1020, 50) mm, rotated rx -180 ry 0 rz 90 deg; joints [-16.626, -86.102, 130.736, 54.303, 12.81, -66.681]
  MoveL 304 to (-351.4, 1020, 50) mm, rotated rx 180 ry 0 rz 90 deg; joints [-14.412, -86.729, 131.417, 51.661, 11.519, -62.387]
  MoveL 305 to (-351.4, 1020, -0.5) mm, rotated rx -180 ry 0 rz 90 deg; joints [-14.412, -84.128, 132.141, 66.894, 9.805, -77.882]
  MoveL 306 to (-351.4, 1020, 50) mm, rotated rx 180 ry 0 rz 90 deg; joints [-14.412, -86.729, 131.417, 51.661, 11.519, -62.387]
  MoveL 307 to (-450, 50, 50) mm, rotated rx -180 ry 0 rz 90 deg; joints [-5.525, -47.552, 74.126, 8.31, 24.786, -11.853]
  MoveL 308 to (-450, 50, -0.5) mm, rotated rx 180 ry 0 rz 90 deg; joints [-5.525, -46.28, 74.665, 8.923, 22.995, -12.523]
  MoveL 309 to (-450, 50, 50) mm, rotated rx -180 ry 0 rz 90 deg; joints [-5.525, -47.552, 74.126, 8.31, 24.786, -11.853]
  MoveL 310 to (-450, 100, 50) mm, rotated rx 180 ry 0 rz 90 deg; joints [-5.655, -49.762, 77.94, 9.05, 23.218, -12.728]
  MoveL 311 to (-450, 100, -0.5) mm, rotated rx -180 ry 0 rz 90 deg; joints [-5.655, -48.445, 78.471, 9.787, 21.394, -13.525]
  MoveL 312 to (-450, 100, 50) mm, rotated rx 180 ry 0 rz 90 deg; joints [-5.655, -49.762, 77.94, 9.05, 23.218, -12.728]
  MoveL 313 to (-450, 150, 50) mm, rotated rx 180 ry 0 rz 90 deg; joints [-5.79, -51.912, 81.605, 9.869, 21.743, -13.685]
  MoveL 314 to (-450, 150, -0.5) mm, rotated rx 180 ry 0 rz 90 deg; joints [-5.79, -50.548, 82.131, 10.759, 19.883, -14.637]
  MoveL 315 to (-450, 150, 50) mm, rotated rx 180 ry 0 rz 90 deg; joints [-5.79, -51.912, 81.605, 9.869, 21.743, -13.685]
  MoveL 316 to (-450, 200, 50) mm, rotated rx 180 ry 0 rz 90 deg; joints [-5.933, -54.012, 85.139, 10.778, 20.353, -14.737]
  MoveL 317 to (-450, 200, -0.5) mm, rotated rx 180 ry 0 rz 90 deg; joints [-5.933, -52.602, 85.663, 11.856, 18.456, -15.879]
  MoveL 318 to (-450, 200, 50) mm, rotated rx 180 ry 0 rz 90 deg; joints [-5.933, -54.012, 85.139, 10.778, 20.353, -14.737]
  MoveL 319 to (-450, 250, 50) mm, rotated rx -180 ry 0 rz 90 deg; joints [-6.082, -56.072, 88.559, 11.791, 19.045, -15.896]
  MoveL 320 to (-450, 250, -0.5) mm, rotated rx -180 ry 0 rz 90 deg; joints [-6.082, -54.613, 89.083, 13.1, 17.109, -17.273]
  MoveL 321 to (-450, 250, 50) mm, rotated rx -180 ry 0 rz 90 deg; joints [-6.082, -56.072, 88.559, 11.791, 19.045, -15.896]
  MoveL 322 to (-450, 300, 50) mm, rotated rx -180 ry 0 rz 90 deg; joints [-6.239, -58.1, 91.877, 12.919, 17.813, -17.175]
  MoveL 323 to (-450, 300, -0.5) mm, rotated rx 180 ry 0 rz 90 deg; joints [-6.239, -56.591, 92.402, 14.514, 15.836, -18.842]
  MoveL 324 to (-450, 300, 50) mm, rotated rx -180 ry 0 rz 90 deg; joints [-6.239, -58.1, 91.877, 12.919, 17.813, -17.175]
  MoveL 325 to (-450, 350, 50) mm, rotated rx 180 ry 0 rz 90 deg; joints [-6.404, -60.104, 95.104, 14.177, 16.655, -18.59]
  MoveL 326 to (-450, 350, -0.5) mm, rotated rx 180 ry 0 rz 90 deg; joints [-6.404, -58.542, 95.632, 16.128, 14.638, -20.616]
  MoveL 327 to (-450, 350, 50) mm, rotated rx 180 ry 0 rz 90 deg; joints [-6.404, -60.104, 95.104, 14.177, 16.655, -18.59]
  MoveL 328 to (-450, 400, 50) mm, rotated rx 180 ry 0 rz 90 deg; joints [-6.579, -62.089, 98.248, 15.58, 15.571, -20.156]
  MoveL 329 to (-450, 400, -0.5) mm, rotated rx -180 ry 0 rz 90 deg; joints [-6.579, -60.472, 98.781, 17.972, 13.513, -22.627]
  MoveL 330 to (-450, 400, 50) mm, rotated rx 180 ry 0 rz 90 deg; joints [-6.579, -62.089, 98.248, 15.58, 15.571, -20.156]
  MoveL 331 to (-450, 450, 50) mm, rotated rx -180 ry 0 rz 90 deg; joints [-6.763, -64.062, 101.318, 17.143, 14.561, -21.889]
  MoveL 332 to (-450, 450, -0.5) mm, rotated rx 180 ry 0 rz 90 deg; joints [-6.763, -62.388, 101.856, 20.084, 12.463, -24.912]
  MoveL 333 to (-450, 450, 50) mm, rotated rx -180 ry 0 rz 90 deg; joints [-6.763, -64.062, 101.318, 17.143, 14.561, -21.889]
  MoveL 334 to (-450, 500, 50) mm, rotated rx -180 ry 0 rz 90 deg; joints [-6.957, -66.03, 104.319, 18.88, 13.626, -23.802]
  MoveL 335 to (-450, 500, -0.5) mm, rotated rx -180 ry 0 rz 90 deg; joints [-6.957, -64.294, 104.865, 22.5, 11.49, -27.51]
  MoveL 336 to (-450, 500, 50) mm, rotated rx -180 ry 0 rz 90 deg; joints [-6.957, -66.03, 104.319, 18.88, 13.626, -23.802]
  MoveL 337 to (-450, 550, 50) mm, rotated rx -180 ry 0 rz 90 deg; joints [-7.163, -67.997, 107.257, 20.801, 12.767, -25.908]
  MoveL 338 to (-450, 550, -0.5) mm, rotated rx 180 ry 0 rz 90 deg; joints [-7.163, -66.197, 107.812, 25.258, 10.598, -30.458]
  MoveL 339 to (-450, 550, 50) mm, rotated rx -180 ry 0 rz 90 deg; joints [-7.163, -67.997, 107.257, 20.801, 12.767, -25.908]
  MoveL 340 to (-450, 600, 50) mm, rotated rx 180 ry 0 rz 90 deg; joints [-7.382, -69.969, 110.136, 22.911, 11.987, -28.211]
  MoveL 341 to (-450, 600, -0.5) mm, rotated rx 180 ry 0 rz 90 deg; joints [-7.382, -68.102, 110.703, 28.391, 9.791, -33.79]
  MoveL 342 to (-450, 600, 50) mm, rotated rx 180 ry 0 rz 90 deg; joints [-7.382, -69.969, 110.136, 22.911, 11.987, -28.211]
  MoveL 343 to (-450, 650, 50) mm, rotated rx 180 ry 0 rz 90 deg; joints [-7.614, -71.954, 112.962, 25.208, 11.291, -30.71]
  MoveL 344 to (-450, 650, -0.5) mm, rotated rx -180 ry 0 rz 90 deg; joints [-7.614, -70.014, 113.541, 31.916, 9.075, -37.524]
  MoveL 345 to (-450, 650, 50) mm, rotated rx 180 ry 0 rz 90 deg; joints [-7.614, -71.954, 112.962, 25.208, 11.291, -30.71]
  MoveL 346 to (-450, 700, 50) mm, rotated rx 180 ry 0 rz 90 deg; joints [-7.861, -73.956, 115.738, 27.673, 10.681, -33.388]
  MoveL 347 to (-450, 700, -0.5) mm, rotated rx 180 ry 0 rz 90 deg; joints [-7.861, -71.94, 116.331, 35.827, 8.456, -41.655]
  MoveL 348 to (-450, 700, 50) mm, rotated rx 180 ry 0 rz 90 deg; joints [-7.861, -73.956, 115.738, 27.673, 10.681, -33.388]
  MoveL 349 to (-450, 750, 50) mm, rotated rx 180 ry 0 rz 90 deg; joints [-8.125, -75.983, 118.466, 30.273, 10.162, -36.211]
  MoveL 350 to (-450, 750, -0.5) mm, rotated rx -180 ry 0 rz 90 deg; joints [-8.125, -73.885, 119.075, 40.076, 7.941, -46.136]
  MoveL 351 to (-450, 750, 50) mm, rotated rx 180 ry 0 rz 90 deg; joints [-8.125, -75.983, 118.466, 30.273, 10.162, -36.211]
  MoveL 352 to (-450, 800, 50) mm, rotated rx 180 ry 0 rz 90 deg; joints [-8.407, -78.043, 121.149, 32.951, 9.739, -39.124]
  MoveL 353 to (-450, 800, -0.5) mm, rotated rx 180 ry 0 rz 90 deg; joints [-8.407, -75.857, 121.777, 44.567, 7.534, -50.87]
  MoveL 354 to (-450, 800, 50) mm, rotated rx 180 ry 0 rz 90 deg; joints [-8.407, -78.043, 121.149, 32.951, 9.739, -39.124]
  MoveL 355 to (-450, 850, 50) mm, rotated rx -180 ry 0 rz 90 deg; joints [-8.709, -80.142, 123.79, 35.626, 9.415, -42.047]
  MoveL 356 to (-450, 850, -0.5) mm, rotated rx -180 ry 0 rz 90 deg; joints [-8.709, -77.863, 124.438, 49.14, 7.238, -55.702]
  MoveL 357 to (-450, 850, 50) mm, rotated rx -180 ry 0 rz 90 deg; joints [-8.709, -80.142, 123.79, 35.626, 9.415, -42.047]
  MoveL 358 to (-450, 900, 50) mm, rotated rx -180 ry 0 rz 90 deg; joints [-9.033, -82.291, 126.39, 38.195, 9.195, -44.879]
  MoveL 359 to (-450, 900, -0.5) mm, rotated rx 180 ry 0 rz 90 deg; joints [-9.033, -79.911, 127.061, 53.588, 7.053, -60.423]
  MoveL 360 to (-450, 900, 50) mm, rotated rx -180 ry 0 rz 90 deg; joints [-9.033, -82.291, 126.39, 38.195, 9.195, -44.879]
  MoveL 361 to (-450, 950, 50) mm, rotated rx 180 ry 0 rz 90 deg; joints [-9.383, -84.5, 128.95, 40.54, 9.082, -47.501]
  MoveL 362 to (-450, 950, -0.5) mm, rotated rx 180 ry 0 rz 90 deg; joints [-9.383, -82.012, 129.647, 57.672, 6.974, -64.797]
  MoveL 363 to (-450, 950, 50) mm, rotated rx 180 ry 0 rz 90 deg; joints [-9.383, -84.5, 128.95, 40.54, 9.082, -47.501]
  MoveL 364 to (-450, 1000, 50) mm, rotated rx 180 ry 0 rz 90 deg; joints [-9.76, -86.78, 131.472, 42.535, 9.079, -49.789]
  MoveL 365 to (-450, 1000, -0.5) mm, rotated rx -180 ry 0 rz 90 deg; joints [-9.76, -84.177, 132.197, 61.157, 6.995, -68.59]
  MoveL 366 to (-450, 1000, 50) mm, rotated rx 180 ry 0 rz 90 deg; joints [-9.76, -86.78, 131.472, 42.535, 9.079, -49.789]
  MoveL 367 to (-450, 1050, 50) mm, rotated rx -180 ry 0 rz 90 deg; joints [-10.168, -89.146, 133.955, 44.06, 9.193, -51.625]
  MoveL 368 to (-450, 1050, -0.5) mm, rotated rx -180 ry 0 rz 90 deg; joints [-10.168, -86.418, 134.713, 63.837, 7.11, -71.597]
  MoveL 369 to (-450, 1050, 50) mm, rotated rx -180 ry 0 rz 90 deg; joints [-10.168, -89.146, 133.955, 44.06, 9.193, -51.625]
  MoveL 370 to (-450, 1100, 50) mm, rotated rx -180 ry 0 rz 90 deg; joints [-10.611, -91.614, 136.401, 45.018, 9.43, -52.912]
  MoveL 371 to (-450, 1100, -0.5) mm, rotated rx -180 ry 0 rz 90 deg; joints [-10.611, -88.752, 137.195, 65.555, 7.313, -73.662]
  MoveL 372 to (-450, 1100, 50) mm, rotated rx -180 ry 0 rz 90 deg; joints [-10.611, -91.614, 136.401, 45.018, 9.43, -52.912]
  MoveL 373 to (-450, 1150, 50) mm, rotated rx 180 ry 0 rz 90 deg; joints [-11.095, -94.203, 138.807, 45.34, 9.803, -53.584]
  MoveL 374 to (-450, 1150, -0.5) mm, rotated rx 180 ry 0 rz 90 deg; joints [-11.095, -91.198, 139.642, 66.205, 7.605, -74.683]
  MoveL 375 to (-450, 1150, 50) mm, rotated rx 180 ry 0 rz 90 deg; joints [-11.095, -94.203, 138.807, 45.34, 9.803, -53.584]
  MoveL 376 to (-450, 1200, 50) mm, rotated rx -180 ry 0 rz 90 deg; joints [-11.624, -96.937, 141.172, 44.999, 10.33, -53.613]
  MoveL 377 to (-450, 1200, -0.5) mm, rotated rx -180 ry 0 rz 90 deg; joints [-11.624, -93.778, 142.054, 65.735, 7.995, -74.607]
  MoveL 378 to (-450, 1200, 50) mm, rotated rx -180 ry 0 rz 90 deg; joints [-11.624, -96.937, 141.172, 44.999, 10.33, -53.613]
  MoveL 379 to (-450, 1250, 50) mm, rotated rx 180 ry 0 rz 90 deg; joints [-12.205, -99.844, 143.495, 44.009, 11.04, -53.016]
  MoveL 380 to (-450, 1250, -0.5) mm, rotated rx 180 ry 0 rz 90 deg; joints [-12.205, -96.52, 144.429, 64.143, 8.502, -73.435]
  MoveL 381 to (-450, 1250, 50) mm, rotated rx 180 ry 0 rz 90 deg; joints [-12.205, -99.844, 143.495, 44.009, 11.04, -53.016]
  MoveL 382 to (-450, 1300, 50) mm, rotated rx 180 ry 0 rz 90 deg; joints [-12.846, -102.957, 145.772, 42.429, 11.969, -51.852]
  MoveL 383 to (-450, 1300, -0.5) mm, rotated rx 180 ry 0 rz 90 deg; joints [-12.846, -99.461, 146.766, 61.485, 9.162, -71.225]
  MoveL 384 to (-450, 1300, 50) mm, rotated rx 180 ry 0 rz 90 deg; joints [-12.846, -102.957, 145.772, 42.429, 11.969, -51.852]
  MoveL 385 to (-450, 1350, 50) mm, rotated rx 180 ry 0 rz 90 deg; joints [-13.557, -106.317, 147.998, 40.357, 13.168, -50.219]
  MoveL 386 to (-450, 1350, -0.5) mm, rotated rx 180 ry 0 rz 90 deg; joints [-13.557, -102.642, 149.061, 57.888, 10.03, -68.103]
  MoveL 387 to (-450, 1350, 50) mm, rotated rx 180 ry 0 rz 90 deg; joints [-13.557, -106.317, 147.998, 40.357, 13.168, -50.219]
  MoveL 388 to (-450, 1400, 50) mm, rotated rx 180 ry 0 rz 90 deg; joints [-14.349, -109.976, 150.167, 37.92, 14.702, -48.244]
  MoveL 389 to (-450, 1400, -0.5) mm, rotated rx 180 ry 0 rz 90 deg; joints [-14.349, -106.121, 151.309, 53.549, 11.18, -64.267]
  MoveL 390 to (-450, 1400, 50) mm, rotated rx 180 ry 0 rz 90 deg; joints [-14.349, -109.976, 150.167, 37.92, 14.702, -48.244]
  MoveL 391 to (-450, 1450, 50) mm, rotated rx 180 ry 0 rz 90 deg; joints [-15.238, -113.994, 152.271, 35.262, 16.649, -46.067]
  MoveL 392 to (-450, 1450, -0.5) mm, rotated rx 180 ry 0 rz 90 deg; joints [-15.238, -109.966, 153.502, 48.732, 12.712, -59.979]
  MoveL 393 to (-450, 1450, 50) mm, rotated rx 180 ry 0 rz 90 deg; joints [-15.238, -113.994, 152.271, 35.262, 16.649, -46.067]
  MoveL 394 to (-578.4, 50, 50) mm, rotated rx -180 ry 0 rz 90 deg; joints [-2.153, -47.939, 74.797, 3.306, 24.197, -4.689]
  MoveL 395 to (-578.4, 50, -0.5) mm, rotated rx 180 ry 0 rz 90 deg; joints [-2.153, -46.659, 75.334, 3.559, 22.383, -4.965]
  MoveL 396 to (-578.4, 50, 50) mm, rotated rx -180 ry 0 rz 90 deg; joints [-2.153, -47.939, 74.797, 3.306, 24.197, -4.689]
  MoveL 397 to (-578.4, 100, 50) mm, rotated rx 180 ry 0 rz 90 deg; joints [-2.203, -50.146, 78.598, 3.608, 22.609, -5.044]
  MoveL 398 to (-578.4, 100, -0.5) mm, rotated rx -180 ry 0 rz 90 deg; joints [-2.203, -48.821, 79.129, 3.914, 20.757, -5.374]
  MoveL 399 to (-578.4, 100, 50) mm, rotated rx 180 ry 0 rz 90 deg; joints [-2.203, -50.146, 78.598, 3.608, 22.609, -5.044]
  MoveL 400 to (-578.4, 150, 50) mm, rotated rx -180 ry 0 rz 90 deg; joints [-2.256, -52.296, 82.254, 3.945, 21.109, -5.435]
  MoveL 401 to (-578.4, 150, -0.5) mm, rotated rx 180 ry 0 rz 90 deg; joints [-2.256, -50.924, 82.78, 4.317, 19.216, -5.832]
  MoveL 402 to (-578.4, 150, 50) mm, rotated rx -180 ry 0 rz 90 deg; joints [-2.256, -52.296, 82.254, 3.945, 21.109, -5.435]
  MoveL 403 to (-578.4, 200, 50) mm, rotated rx 180 ry 0 rz 90 deg; joints [-2.312, -54.397, 85.783, 4.322, 19.689, -5.867]
  MoveL 404 to (-578.4, 200, -0.5) mm, rotated rx -180 ry 0 rz 90 deg; joints [-2.312, -52.978, 86.306, 4.777, 17.752, -6.348]
  MoveL 405 to (-578.4, 200, 50) mm, rotated rx 180 ry 0 rz 90 deg; joints [-2.312, -54.397, 85.783, 4.322, 19.689, -5.867]
  MoveL 406 to (-578.4, 250, 50) mm, rotated rx 180 ry 0 rz 90 deg; joints [-2.371, -56.46, 89.199, 4.745, 18.345, -6.347]
  MoveL 407 to (-578.4, 250, -0.5) mm, rotated rx 180 ry 0 rz 90 deg; joints [-2.371, -54.992, 89.722, 5.303, 16.36, -6.932]
  MoveL 408 to (-578.4, 250, 50) mm, rotated rx 180 ry 0 rz 90 deg; joints [-2.371, -56.46, 89.199, 4.745, 18.345, -6.347]
  MoveL 409 to (-578.4, 300, 50) mm, rotated rx 180 ry 0 rz 90 deg; joints [-2.432, -58.493, 92.515, 5.22, 17.071, -6.882]
  MoveL 410 to (-578.4, 300, -0.5) mm, rotated rx -180 ry 0 rz 90 deg; joints [-2.432, -56.974, 93.04, 5.91, 15.035, -7.599]
  MoveL 411 to (-578.4, 300, 50) mm, rotated rx 180 ry 0 rz 90 deg; joints [-2.432, -58.493, 92.515, 5.22, 17.071, -6.882]
  MoveL 412 to (-578.4, 350, 50) mm, rotated rx 180 ry 0 rz 90 deg; joints [-2.497, -60.503, 95.741, 5.757, 15.865, -7.481]
  MoveL 413 to (-578.4, 350, -0.5) mm, rotated rx 180 ry 0 rz 90 deg; joints [-2.497, -58.931, 96.27, 6.613, 13.775, -8.366]
  MoveL 414 to (-578.4, 350, 50) mm, rotated rx 180 ry 0 rz 90 deg; joints [-2.497, -60.503, 95.741, 5.757, 15.865, -7.481]
  MoveL 415 to (-578.4, 400, 50) mm, rotated rx -180 ry 0 rz 90 deg; joints [-2.566, -62.497, 98.887, 6.364, 14.724, -8.151]
  MoveL 416 to (-578.4, 400, -0.5) mm, rotated rx 180 ry 0 rz 90 deg; joints [-2.566, -60.868, 99.421, 7.433, 12.578, -9.252]
  MoveL 417 to (-578.4, 400, 50) mm, rotated rx -180 ry 0 rz 90 deg; joints [-2.566, -62.497, 98.887, 6.364, 14.724, -8.151]
  MoveL 418 to (-578.4, 450, 50) mm, rotated rx 180 ry 0 rz 90 deg; joints [-2.638, -64.48, 101.96, 7.051, 13.649, -8.905]
  MoveL 419 to (-578.4, 450, -0.5) mm, rotated rx 180 ry 0 rz 90 deg; joints [-2.638, -62.793, 102.5, 8.396, 11.442, -10.283]
  MoveL 420 to (-578.4, 450, 50) mm, rotated rx 180 ry 0 rz 90 deg; joints [-2.638, -64.48, 101.96, 7.051, 13.649, -8.905]
  MoveL 421 to (-578.4, 500, 50) mm, rotated rx -180 ry 0 rz 90 deg; joints [-2.715, -66.459, 104.965, 7.829, 12.639, -9.752]
  MoveL 422 to (-578.4, 500, -0.5) mm, rotated rx 180 ry 0 rz 90 deg; joints [-2.715, -64.71, 105.513, 9.533, 10.368, -11.491]
  MoveL 423 to (-578.4, 500, 50) mm, rotated rx -180 ry 0 rz 90 deg; joints [-2.715, -66.459, 104.965, 7.829, 12.639, -9.752]
  MoveL 424 to (-578.4, 550, 50) mm, rotated rx -180 ry 0 rz 90 deg; joints [-2.796, -68.439, 107.909, 8.71, 11.695, -10.706]
  MoveL 425 to (-578.4, 550, -0.5) mm, rotated rx 180 ry 0 rz 90 deg; joints [-2.796, -66.625, 108.467, 10.883, 9.357, -12.915]
  MoveL 426 to (-578.4, 550, 50) mm, rotated rx -180 ry 0 rz 90 deg; joints [-2.796, -68.439, 107.909, 8.71, 11.695, -10.706]
  MoveL 427 to (-578.4, 600, 50) mm, rotated rx 180 ry 0 rz 90 deg; joints [-2.882, -70.428, 110.796, 9.705, 10.819, -11.776]
  MoveL 428 to (-578.4, 600, -0.5) mm, rotated rx 180 ry 0 rz 90 deg; joints [-2.882, -68.544, 111.365, 12.493, 8.411, -14.603]
  MoveL 429 to (-578.4, 600, 50) mm, rotated rx 180 ry 0 rz 90 deg; joints [-2.882, -70.428, 110.796, 9.705, 10.819, -11.776]
  MoveL 430 to (-578.4, 650, 50) mm, rotated rx -180 ry 0 rz 90 deg; joints [-2.974, -72.431, 113.631, 10.823, 10.012, -12.973]
  MoveL 431 to (-578.4, 650, -0.5) mm, rotated rx -180 ry 0 rz 90 deg; joints [-2.974, -70.473, 114.213, 14.419, 7.533, -16.612]
  MoveL 432 to (-578.4, 650, 50) mm, rotated rx -180 ry 0 rz 90 deg; joints [-2.974, -72.431, 113.631, 10.823, 10.012, -12.973]
  MoveL 433 to (-578.4, 700, 50) mm, rotated rx -180 ry 0 rz 90 deg; joints [-3.071, -74.455, 116.416, 12.068, 9.28, -14.302]
  MoveL 434 to (-578.4, 700, -0.5) mm, rotated rx -180 ry 0 rz 90 deg; joints [-3.071, -72.419, 117.013, 16.726, 6.728, -19.005]
  MoveL 435 to (-578.4, 700, 50) mm, rotated rx -180 ry 0 rz 90 deg; joints [-3.071, -74.455, 116.416, 12.068, 9.28, -14.302]
  MoveL 436 to (-578.4, 750, 50) mm, rotated rx 180 ry 0 rz 90 deg; joints [-3.175, -76.506, 119.156, 13.439, 8.626, -15.761]
  MoveL 437 to (-578.4, 750, -0.5) mm, rotated rx -180 ry 0 rz 90 deg; joints [-3.175, -74.386, 119.77, 19.477, 6.001, -21.847]
  MoveL 438 to (-578.4, 750, 50) mm, rotated rx 180 ry 0 rz 90 deg; joints [-3.175, -76.506, 119.156, 13.439, 8.626, -15.761]
  MoveL 439 to (-578.4, 800, 50) mm, rotated rx 180 ry 0 rz 90 deg; joints [-3.287, -78.594, 121.852, 14.92, 8.056, -17.334]
  MoveL 440 to (-578.4, 800, -0.5) mm, rotated rx 180 ry 0 rz 90 deg; joints [-3.287, -76.384, 122.485, 22.724, 5.359, -25.19]
  MoveL 441 to (-578.4, 800, 50) mm, rotated rx 180 ry 0 rz 90 deg; joints [-3.287, -78.594, 121.852, 14.92, 8.056, -17.334]
  MoveL 442 to (-578.4, 850, 50) mm, rotated rx 180 ry 0 rz 90 deg; joints [-3.406, -80.727, 124.508, 16.476, 7.576, -18.988]
  MoveL 443 to (-578.4, 850, -0.5) mm, rotated rx -180 ry 0 rz 90 deg; joints [-3.406, -78.421, 125.161, 26.476, 4.811, -29.044]
  MoveL 444 to (-578.4, 850, 50) mm, rotated rx 180 ry 0 rz 90 deg; joints [-3.406, -80.727, 124.508, 16.476, 7.576, -18.988]
  MoveL 445 to (-578.4, 900, 50) mm, rotated rx 180 ry 0 rz 90 deg; joints [-3.535, -82.914, 127.124, 18.05, 7.194, -20.666]
  MoveL 446 to (-578.4, 900, -0.5) mm, rotated rx -180 ry 0 rz 90 deg; joints [-3.535, -80.504, 127.801, 30.656, 4.364, -33.332]
  MoveL 447 to (-578.4, 900, 50) mm, rotated rx 180 ry 0 rz 90 deg; joints [-3.535, -82.914, 127.124, 18.05, 7.194, -20.666]
  MoveL 448 to (-578.4, 950, 50) mm, rotated rx 180 ry 0 rz 90 deg; joints [-3.674, -85.167, 129.702, 19.556, 6.919, -22.281]
  MoveL 449 to (-578.4, 950, -0.5) mm, rotated rx 180 ry 0 rz 90 deg; joints [-3.674, -82.647, 130.406, 35.049, 4.026, -37.839]
  MoveL 450 to (-578.4, 950, 50) mm, rotated rx 180 ry 0 rz 90 deg; joints [-3.674, -85.167, 129.702, 19.556, 6.919, -22.281]
  MoveL 451 to (-578.4, 1000, 50) mm, rotated rx -180 ry 0 rz 90 deg; joints [-3.824, -87.5, 132.243, 20.885, 6.761, -23.725]
  MoveL 452 to (-578.4, 1000, -0.5) mm, rotated rx 180 ry 0 rz 90 deg; joints [-3.824, -84.86, 132.977, 39.27, 3.802, -42.182]
  MoveL 453 to (-578.4, 1000, 50) mm, rotated rx -180 ry 0 rz 90 deg; joints [-3.824, -87.5, 132.243, 20.885, 6.761, -23.725]
  MoveL 454 to (-578.4, 1050, 50) mm, rotated rx 180 ry 0 rz 90 deg; joints [-3.986, -89.929, 134.747, 21.914, 6.732, -24.878]
  MoveL 455 to (-578.4, 1050, -0.5) mm, rotated rx 180 ry 0 rz 90 deg; joints [-3.986, -87.159, 135.516, 42.798, 3.692, -45.838]
  MoveL 456 to (-578.4, 1050, 50) mm, rotated rx 180 ry 0 rz 90 deg; joints [-3.986, -89.929, 134.747, 21.914, 6.732, -24.878]
  MoveL 457 to (-578.4, 1100, 50) mm, rotated rx 180 ry 0 rz 90 deg; joints [-4.164, -92.471, 137.215, 22.531, 6.848, -25.624]
  MoveL 458 to (-578.4, 1100, -0.5) mm, rotated rx -180 ry 0 rz 90 deg; joints [-4.164, -89.562, 138.022, 45.086, 3.699, -48.264]
  MoveL 459 to (-578.4, 1100, 50) mm, rotated rx 180 ry 0 rz 90 deg; joints [-4.164, -92.471, 137.215, 22.531, 6.848, -25.624]
  MoveL 460 to (-578.4, 1150, 50) mm, rotated rx 180 ry 0 rz 90 deg; joints [-4.357, -95.149, 139.645, 22.656, 7.13, -25.887]
  MoveL 461 to (-578.4, 1150, -0.5) mm, rotated rx 180 ry 0 rz 90 deg; joints [-4.357, -92.091, 140.496, 45.719, 3.829, -49.044]
  MoveL 462 to (-578.4, 1150, 50) mm, rotated rx 180 ry 0 rz 90 deg; joints [-4.357, -95.149, 139.645, 22.656, 7.13, -25.887]
  MoveL 463 to (-578.4, 1200, 50) mm, rotated rx -180 ry 0 rz 90 deg; joints [-4.57, -97.991, 142.037, 22.265, 7.604, -25.643]
  MoveL 464 to (-578.4, 1200, -0.5) mm, rotated rx 180 ry 0 rz 90 deg; joints [-4.57, -94.772, 142.937, 44.543, 4.099, -48.024]
  MoveL 465 to (-578.4, 1200, 50) mm, rotated rx -180 ry 0 rz 90 deg; joints [-4.57, -97.991, 142.037, 22.265, 7.604, -25.643]
  MoveL 466 to (-578.4, 1250, 50) mm, rotated rx -180 ry 0 rz 90 deg; joints [-4.804, -101.03, 144.388, 21.398, 8.306, -24.931]
  MoveL 467 to (-578.4, 1250, -0.5) mm, rotated rx 180 ry 0 rz 90 deg; joints [-4.804, -97.64, 145.344, 41.715, 4.543, -45.362]
  MoveL 468 to (-578.4, 1250, 50) mm, rotated rx -180 ry 0 rz 90 deg; joints [-4.804, -101.03, 144.388, 21.398, 8.306, -24.931]
  MoveL 469 to (-578.4, 1300, 50) mm, rotated rx 180 ry 0 rz 90 deg; joints [-5.064, -104.306, 146.694, 20.147, 9.281, -23.843]
  MoveL 470 to (-578.4, 1300, -0.5) mm, rotated rx -180 ry 0 rz 90 deg; joints [-5.064, -100.737, 147.715, 37.674, 5.214, -41.499]
  MoveL 471 to (-578.4, 1300, 50) mm, rotated rx 180 ry 0 rz 90 deg; joints [-5.064, -104.306, 146.694, 20.147, 9.281, -23.843]
  MoveL 472 to (-578.4, 1350, 50) mm, rotated rx 180 ry 0 rz 90 deg; joints [-5.353, -107.87, 148.95, 18.636, 10.586, -22.505]
  MoveL 473 to (-578.4, 1350, -0.5) mm, rotated rx 180 ry 0 rz 90 deg; joints [-5.353, -104.117, 150.045, 33.01, 6.186, -37.022]
  MoveL 474 to (-578.4, 1350, 50) mm, rotated rx 180 ry 0 rz 90 deg; joints [-5.353, -107.87, 148.95, 18.636, 10.586, -22.505]
  MoveL 475 to (-578.4, 1400, 50) mm, rotated rx 180 ry 0 rz 90 deg; joints [-5.677, -111.786, 151.149, 16.996, 12.296, -21.045]
  MoveL 476 to (-578.4, 1400, -0.5) mm, rotated rx 180 ry 0 rz 90 deg; joints [-5.677, -107.85, 152.331, 28.283, 7.549, -32.492]
  MoveL 477 to (-578.4, 1400, 50) mm, rotated rx 180 ry 0 rz 90 deg; joints [-5.677, -111.786, 151.149, 16.996, 12.296, -21.045]
  MoveL 478 to (-578.4, 1450, 50) mm, rotated rx -180 ry 0 rz 90 deg; joints [-6.042, -116.131, 153.282, 15.34, 14.501, -19.576]
  MoveL 479 to (-578.4, 1450, -0.5) mm, rotated rx -180 ry 0 rz 90 deg; joints [-6.042, -112.026, 154.563, 23.892, 9.413, -28.308]
  MoveL 480 to (-578.4, 1450, 50) mm, rotated rx -180 ry 0 rz 90 deg; joints [-6.042, -116.131, 153.282, 15.34, 14.501, -19.576]
  MoveL 481 to (-476, 1150, 50) mm, rotated rx -180 ry 0 rz 90 deg; joints [-9.749, -94.459, 139.035, 42.023, 9.16, -49.264]
  MoveL 482 to (-476, 1150, -0.5) mm, rotated rx 180 ry 0 rz 90 deg; joints [-9.749, -91.439, 139.874, 64.189, 6.798, -71.635]
  MoveL 483 to (-476, 1150, 50) mm, rotated rx -180 ry 0 rz 90 deg; joints [-9.749, -94.459, 139.035, 42.023, 9.16, -49.264]
  MoveL 484 to (-514.2, 1150, 50) mm, rotated rx 180 ry 0 rz 90 deg; joints [-7.753, -94.776, 139.317, 36.075, 8.29, -41.829]
  MoveL 485 to (-514.2, 1150, -0.5) mm, rotated rx -180 ry 0 rz 90 deg; joints [-7.753, -91.739, 140.162, 59.875, 5.633, -65.794]
  MoveL 486 to (-514.2, 1150, 50) mm, rotated rx 180 ry 0 rz 90 deg; joints [-7.753, -94.776, 139.317, 36.075, 8.29, -41.829]
  MoveL 487 to (-552.4, 1150, 50) mm, rotated rx 180 ry 0 rz 90 deg; joints [-5.738, -95.023, 139.534, 28.638, 7.543, -32.893]
  MoveL 488 to (-552.4, 1150, -0.5) mm, rotated rx -180 ry 0 rz 90 deg; joints [-5.738, -91.971, 140.383, 52.939, 4.522, -57.318]
  MoveL 489 to (-552.4, 1150, 50) mm, rotated rx 180 ry 0 rz 90 deg; joints [-5.738, -95.023, 139.534, 28.638, 7.543, -32.893]
  MoveL 490 to (-655, 50, 50) mm, rotated rx 180 ry 0 rz 90 deg; joints [-0.132, -48.007, 74.916, 0.203, 24.092, -0.288]
  MoveL 491 to (-655, 50, -0.5) mm, rotated rx 180 ry 0 rz 90 deg; joints [-0.132, -46.726, 75.453, 0.219, 22.274, -0.305]
  MoveL 492 to (-655, 50, 50) mm, rotated rx 180 ry 0 rz 90 deg; joints [-0.132, -48.007, 74.916, 0.203, 24.092, -0.288]
  MoveL 493 to (-655, 100, 50) mm, rotated rx -180 ry 0 rz 90 deg; joints [-0.135, -50.215, 78.715, 0.222, 22.5, -0.31]
  MoveL 494 to (-655, 100, -0.5) mm, rotated rx -180 ry 0 rz 90 deg; joints [-0.135, -48.888, 79.245, 0.241, 20.643, -0.331]
  MoveL 495 to (-655, 100, 50) mm, rotated rx -180 ry 0 rz 90 deg; joints [-0.135, -50.215, 78.715, 0.222, 22.5, -0.31]
  MoveL 496 to (-655, 150, 50) mm, rotated rx 180 ry 0 rz 90 deg; joints [-0.138, -52.364, 82.369, 0.243, 20.995, -0.334]
  MoveL 497 to (-655, 150, -0.5) mm, rotated rx -180 ry 0 rz 90 deg; joints [-0.138, -50.99, 82.895, 0.266, 19.096, -0.359]
  MoveL 498 to (-655, 150, 50) mm, rotated rx 180 ry 0 rz 90 deg; joints [-0.138, -52.364, 82.369, 0.243, 20.995, -0.334]
  MoveL 499 to (-655, 200, 50) mm, rotated rx -180 ry 0 rz 90 deg; joints [-0.142, -54.466, 85.896, 0.266, 19.569, -0.361]
  MoveL 500 to (-655, 200, -0.5) mm, rotated rx -180 ry 0 rz 90 deg; joints [-0.142, -53.045, 86.42, 0.295, 17.625, -0.391]
  MoveL 501 to (-655, 200, 50) mm, rotated rx -180 ry 0 rz 90 deg; joints [-0.142, -54.466, 85.896, 0.266, 19.569, -0.361]
  MoveL 502 to (-655, 250, 50) mm, rotated rx -180 ry 0 rz 90 deg; joints [-0.145, -56.529, 89.312, 0.293, 18.218, -0.391]
  MoveL 503 to (-655, 250, -0.5) mm, rotated rx -180 ry 0 rz 90 deg; joints [-0.145, -55.059, 89.836, 0.327, 16.224, -0.427]
  MoveL 504 to (-655, 250, 50) mm, rotated rx -180 ry 0 rz 90 deg; joints [-0.145, -56.529, 89.312, 0.293, 18.218, -0.391]
  MoveL 505 to (-655, 300, 50) mm, rotated rx -180 ry 0 rz 90 deg; joints [-0.149, -58.563, 92.628, 0.322, 16.936, -0.424]
  MoveL 506 to (-655, 300, -0.5) mm, rotated rx 180 ry 0 rz 90 deg; joints [-0.149, -57.042, 93.153, 0.365, 14.889, -0.469]
  MoveL 507 to (-655, 300, 50) mm, rotated rx -180 ry 0 rz 90 deg; joints [-0.149, -58.563, 92.628, 0.322, 16.936, -0.424]
  MoveL 508 to (-655, 350, 50) mm, rotated rx 180 ry 0 rz 90 deg; joints [-0.153, -60.574, 95.854, 0.356, 15.72, -0.461]
  MoveL 509 to (-655, 350, -0.5) mm, rotated rx -180 ry 0 rz 90 deg; joints [-0.153, -59, 96.383, 0.409, 13.617, -0.517]
  MoveL 510 to (-655, 350, 50) mm, rotated rx 180 ry 0 rz 90 deg; joints [-0.153, -60.574, 95.854, 0.356, 15.72, -0.461]
  MoveL 511 to (-655, 400, 50) mm, rotated rx -180 ry 0 rz 90 deg; joints [-0.157, -62.569, 99, 0.394, 14.569, -0.503]
  MoveL 512 to (-655, 400, -0.5) mm, rotated rx 180 ry 0 rz 90 deg; joints [-0.157, -60.938, 99.534, 0.461, 12.405, -0.572]
  MoveL 513 to (-655, 400, 50) mm, rotated rx -180 ry 0 rz 90 deg; joints [-0.157, -62.569, 99, 0.394, 14.569, -0.503]
  MoveL 514 to (-655, 450, 50) mm, rotated rx -180 ry 0 rz 90 deg; joints [-0.162, -64.554, 102.073, 0.437, 13.481, -0.55]
  MoveL 515 to (-655, 450, -0.5) mm, rotated rx -180 ry 0 rz 90 deg; joints [-0.162, -62.864, 102.614, 0.522, 11.251, -0.637]
  MoveL 516 to (-655, 450, 50) mm, rotated rx -180 ry 0 rz 90 deg; joints [-0.162, -64.554, 102.073, 0.437, 13.481, -0.55]
  MoveL 517 to (-655, 500, 50) mm, rotated rx -180 ry 0 rz 90 deg; joints [-0.166, -66.535, 105.08, 0.486, 12.456, -0.604]
  MoveL 518 to (-655, 500, -0.5) mm, rotated rx 180 ry 0 rz 90 deg; joints [-0.166, -64.783, 105.628, 0.594, 10.156, -0.714]
  MoveL 519 to (-655, 500, 50) mm, rotated rx -180 ry 0 rz 90 deg; joints [-0.166, -66.535, 105.08, 0.486, 12.456, -0.604]
  MoveL 520 to (-655, 550, 50) mm, rotated rx -180 ry 0 rz 90 deg; joints [-0.171, -68.518, 108.025, 0.541, 11.494, -0.664]
  MoveL 521 to (-655, 550, -0.5) mm, rotated rx -180 ry 0 rz 90 deg; joints [-0.171, -66.701, 108.583, 0.681, 9.119, -0.805]
  MoveL 522 to (-655, 550, 50) mm, rotated rx -180 ry 0 rz 90 deg; joints [-0.171, -68.518, 108.025, 0.541, 11.494, -0.664]
  MoveL 523 to (-655, 600, 50) mm, rotated rx 180 ry 0 rz 90 deg; joints [-0.177, -70.51, 110.913, 0.605, 10.597, -0.732]
  MoveL 524 to (-655, 600, -0.5) mm, rotated rx -180 ry 0 rz 90 deg; joints [-0.177, -68.623, 111.483, 0.785, 8.141, -0.915]
  MoveL 525 to (-655, 600, 50) mm, rotated rx 180 ry 0 rz 90 deg; joints [-0.177, -70.51, 110.913, 0.605, 10.597, -0.732]
  MoveL 526 to (-655, 650, 50) mm, rotated rx -180 ry 0 rz 90 deg; joints [-0.182, -72.516, 113.75, 0.677, 9.767, -0.808]
  MoveL 527 to (-655, 650, -0.5) mm, rotated rx -180 ry 0 rz 90 deg; joints [-0.182, -70.555, 114.332, 0.913, 7.224, -1.047]
  MoveL 528 to (-655, 650, 50) mm, rotated rx -180 ry 0 rz 90 deg; joints [-0.182, -72.516, 113.75, 0.677, 9.767, -0.808]
  MoveL 529 to (-655, 700, 50) mm, rotated rx 180 ry 0 rz 90 deg; joints [-0.188, -74.544, 116.537, 0.757, 9.008, -0.894]
  MoveL 530 to (-655, 700, -0.5) mm, rotated rx -180 ry 0 rz 90 deg; joints [-0.188, -72.504, 117.134, 1.068, 6.371, -1.208]
  MoveL 531 to (-655, 700, 50) mm, rotated rx 180 ry 0 rz 90 deg; joints [-0.188, -74.544, 116.537, 0.757, 9.008, -0.894]
  MoveL 532 to (-655, 750, 50) mm, rotated rx 180 ry 0 rz 90 deg; joints [-0.195, -76.6, 119.279, 0.847, 8.322, -0.989]
  MoveL 533 to (-655, 750, -0.5) mm, rotated rx 180 ry 0 rz 90 deg; joints [-0.195, -74.476, 119.893, 1.26, 5.584, -1.405]
  MoveL 534 to (-655, 750, 50) mm, rotated rx 180 ry 0 rz 90 deg; joints [-0.195, -76.6, 119.279, 0.847, 8.322, -0.989]
  MoveL 535 to (-655, 800, 50) mm, rotated rx -180 ry 0 rz 90 deg; joints [-0.202, -78.693, 121.977, 0.945, 7.716, -1.093]
  MoveL 536 to (-655, 800, -0.5) mm, rotated rx 180 ry 0 rz 90 deg; joints [-0.202, -76.479, 122.611, 1.495, 4.87, -1.646]
  MoveL 537 to (-655, 800, 50) mm, rotated rx -180 ry 0 rz 90 deg; joints [-0.202, -78.693, 121.977, 0.945, 7.716, -1.093]
  MoveL 538 to (-655, 850, 50) mm, rotated rx -180 ry 0 rz 90 deg; joints [-0.209, -80.831, 124.635, 1.05, 7.197, -1.204]
  MoveL 539 to (-655, 850, -0.5) mm, rotated rx -180 ry 0 rz 90 deg; joints [-0.209, -78.52, 125.29, 1.782, 4.232, -1.94]
  MoveL 540 to (-655, 850, 50) mm, rotated rx -180 ry 0 rz 90 deg; joints [-0.209, -80.831, 124.635, 1.05, 7.197, -1.204]
  MoveL 541 to (-655, 900, 50) mm, rotated rx -180 ry 0 rz 90 deg; joints [-0.217, -83.025, 127.254, 1.157, 6.773, -1.318]
  MoveL 542 to (-655, 900, -0.5) mm, rotated rx 180 ry 0 rz 90 deg; joints [-0.217, -80.611, 127.933, 2.127, 3.68, -2.291]
  MoveL 543 to (-655, 900, 50) mm, rotated rx -180 ry 0 rz 90 deg; joints [-0.217, -83.025, 127.254, 1.157, 6.773, -1.318]
  MoveL 544 to (-655, 950, 50) mm, rotated rx -180 ry 0 rz 90 deg; joints [-0.225, -85.287, 129.835, 1.262, 6.454, -1.429]
  MoveL 545 to (-655, 950, -0.5) mm, rotated rx -180 ry 0 rz 90 deg; joints [-0.225, -82.76, 130.541, 2.524, 3.222, -2.696]
  MoveL 546 to (-655, 950, 50) mm, rotated rx -180 ry 0 rz 90 deg; joints [-0.225, -85.287, 129.835, 1.262, 6.454, -1.429]
  MoveL 547 to (-655, 1000, 50) mm, rotated rx -180 ry 0 rz 90 deg; joints [-0.235, -87.63, 132.38, 1.356, 6.252, -1.53]
  MoveL 548 to (-655, 1000, -0.5) mm, rotated rx 180 ry 0 rz 90 deg; joints [-0.235, -84.982, 133.116, 2.95, 2.87, -3.129]
  MoveL 549 to (-655, 1000, 50) mm, rotated rx -180 ry 0 rz 90 deg; joints [-0.235, -87.63, 132.38, 1.356, 6.252, -1.53]
  MoveL 550 to (-655, 1050, 50) mm, rotated rx 180 ry 0 rz 90 deg; joints [-0.245, -90.07, 134.888, 1.429, 6.184, -1.611]
  MoveL 551 to (-655, 1050, -0.5) mm, rotated rx 180 ry 0 rz 90 deg; joints [-0.245, -87.292, 135.659, 3.347, 2.638, -3.534]
  MoveL 552 to (-655, 1050, 50) mm, rotated rx 180 ry 0 rz 90 deg; joints [-0.245, -90.07, 134.888, 1.429, 6.184, -1.611]
  MoveL 553 to (-655, 1100, 50) mm, rotated rx 180 ry 0 rz 90 deg; joints [-0.256, -92.625, 137.36, 1.473, 6.268, -1.663]
  MoveL 554 to (-655, 1100, -0.5) mm, rotated rx -180 ry 0 rz 90 deg; joints [-0.256, -89.708, 138.17, 3.626, 2.544, -3.821]
  MoveL 555 to (-655, 1100, 50) mm, rotated rx 180 ry 0 rz 90 deg; joints [-0.256, -92.625, 137.36, 1.473, 6.268, -1.663]
  MoveL 556 to (-655, 1150, 50) mm, rotated rx 180 ry 0 rz 90 deg; joints [-0.268, -95.32, 139.795, 1.481, 6.528, -1.679]
  MoveL 557 to (-655, 1150, -0.5) mm, rotated rx 180 ry 0 rz 90 deg; joints [-0.268, -92.252, 140.648, 3.7, 2.609, -3.904]
  MoveL 558 to (-655, 1150, 50) mm, rotated rx 180 ry 0 rz 90 deg; joints [-0.268, -95.32, 139.795, 1.481, 6.528, -1.679]
  MoveL 559 to (-655, 1200, 50) mm, rotated rx 180 ry 0 rz 90 deg; joints [-0.281, -98.182, 142.191, 1.45, 6.994, -1.658]
  MoveL 560 to (-655, 1200, -0.5) mm, rotated rx 180 ry 0 rz 90 deg; joints [-0.281, -94.953, 143.095, 3.537, 2.863, -3.751]
  MoveL 561 to (-655, 1200, 50) mm, rotated rx 180 ry 0 rz 90 deg; joints [-0.281, -98.182, 142.191, 1.45, 6.994, -1.658]
  MoveL 562 to (-655, 1250, 50) mm, rotated rx 180 ry 0 rz 90 deg; joints [-0.295, -101.246, 144.547, 1.386, 7.701, -1.603]
  MoveL 563 to (-655, 1250, -0.5) mm, rotated rx -180 ry 0 rz 90 deg; joints [-0.295, -97.844, 145.508, 3.187, 3.342, -3.411]
  MoveL 564 to (-655, 1250, 50) mm, rotated rx 180 ry 0 rz 90 deg; joints [-0.295, -101.246, 144.547, 1.386, 7.701, -1.603]
  MoveL 565 to (-783.4, 50, 50) mm, rotated rx -180 ry 0 rz 90 deg; joints [3.253, -47.851, 74.644, -4.972, 24.333, 7.062]
  MoveL 566 to (-783.4, 50, -0.5) mm, rotated rx 180 ry 0 rz 90 deg; joints [3.253, -46.572, 75.181, -5.35, 22.524, 7.473]
  MoveL 567 to (-783.4, 50, 50) mm, rotated rx -180 ry 0 rz 90 deg; joints [3.253, -47.851, 74.644, -4.972, 24.333, 7.062]
  MoveL 568 to (-783.4, 100, 50) mm, rotated rx 180 ry 0 rz 90 deg; joints [3.33, -50.059, 78.448, -5.424, 22.749, 7.593]
  MoveL 569 to (-783.4, 100, -0.5) mm, rotated rx 180 ry 0 rz 90 deg; joints [3.33, -48.735, 78.978, -5.88, 20.904, 8.084]
  MoveL 570 to (-783.4, 100, 50) mm, rotated rx 180 ry 0 rz 90 deg; joints [3.33, -50.059, 78.448, -5.424, 22.749, 7.593]
  MoveL 571 to (-783.4, 150, 50) mm, rotated rx -180 ry 0 rz 90 deg; joints [3.41, -52.208, 82.106, -5.927, 21.255, 8.178]
  MoveL 572 to (-783.4, 150, -0.5) mm, rotated rx 180 ry 0 rz 90 deg; joints [3.41, -50.838, 82.632, -6.48, 19.37, 8.768]
  MoveL 573 to (-783.4, 150, 50) mm, rotated rx -180 ry 0 rz 90 deg; joints [3.41, -52.208, 82.106, -5.927, 21.255, 8.178]
  MoveL 574 to (-783.4, 200, 50) mm, rotated rx 180 ry 0 rz 90 deg; joints [3.494, -54.309, 85.635, -6.488, 19.843, 8.823]
  MoveL 575 to (-783.4, 200, -0.5) mm, rotated rx -180 ry 0 rz 90 deg; joints [3.494, -52.892, 86.159, -7.163, 17.916, 9.536]
  MoveL 576 to (-783.4, 200, 50) mm, rotated rx 180 ry 0 rz 90 deg; joints [3.494, -54.309, 85.635, -6.488, 19.843, 8.823]
  MoveL 577 to (-783.4, 250, 50) mm, rotated rx -180 ry 0 rz 90 deg; joints [3.583, -56.372, 89.052, -7.117, 18.507, 9.538]
  MoveL 578 to (-783.4, 250, -0.5) mm, rotated rx 180 ry 0 rz 90 deg; joints [3.583, -54.905, 89.576, -7.943, 16.534, 10.404]
  MoveL 579 to (-783.4, 250, 50) mm, rotated rx -180 ry 0 rz 90 deg; joints [3.583, -56.372, 89.052, -7.117, 18.507, 9.538]
  MoveL 580 to (-783.4, 300, 50) mm, rotated rx 180 ry 0 rz 90 deg; joints [3.676, -58.403, 92.369, -7.822, 17.243, 10.333]
  MoveL 581 to (-783.4, 300, -0.5) mm, rotated rx 180 ry 0 rz 90 deg; joints [3.676, -56.886, 92.894, -8.839, 15.222, 11.391]
  MoveL 582 to (-783.4, 300, 50) mm, rotated rx 180 ry 0 rz 90 deg; joints [3.676, -58.403, 92.369, -7.822, 17.243, 10.333]
  MoveL 583 to (-783.4, 350, 50) mm, rotated rx 180 ry 0 rz 90 deg; joints [3.774, -60.412, 95.596, -8.616, 16.049, 11.22]
  MoveL 584 to (-783.4, 350, -0.5) mm, rotated rx 180 ry 0 rz 90 deg; joints [3.774, -58.841, 96.124, -9.874, 13.977, 12.521]
  MoveL 585 to (-783.4, 350, 50) mm, rotated rx 180 ry 0 rz 90 deg; joints [3.774, -60.412, 95.596, -8.616, 16.049, 11.22]
  MoveL 586 to (-783.4, 400, 50) mm, rotated rx 180 ry 0 rz 90 deg; joints [3.877, -62.403, 98.741, -9.511, 14.923, 12.211]
  MoveL 587 to (-783.4, 400, -0.5) mm, rotated rx 180 ry 0 rz 90 deg; joints [3.877, -60.777, 99.274, -11.075, 12.798, 13.821]
  MoveL 588 to (-783.4, 400, 50) mm, rotated rx 180 ry 0 rz 90 deg; joints [3.877, -62.403, 98.741, -9.511, 14.923, 12.211]
  MoveL 589 to (-783.4, 450, 50) mm, rotated rx 180 ry 0 rz 90 deg; joints [3.986, -64.384, 101.813, -10.52, 13.863, 13.319]
  MoveL 590 to (-783.4, 450, -0.5) mm, rotated rx 180 ry 0 rz 90 deg; joints [3.986, -62.7, 102.352, -12.475, 11.684, 15.324]
  MoveL 591 to (-783.4, 450, 50) mm, rotated rx 180 ry 0 rz 90 deg; joints [3.986, -64.384, 101.813, -10.52, 13.863, 13.319]
  MoveL 592 to (-783.4, 500, 50) mm, rotated rx 180 ry 0 rz 90 deg; joints [4.101, -66.36, 104.817, -11.657, 12.872, 14.561]
  MoveL 593 to (-783.4, 500, -0.5) mm, rotated rx 180 ry 0 rz 90 deg; joints [4.101, -64.614, 105.365, -14.115, 10.636, 17.072]
  MoveL 594 to (-783.4, 500, 50) mm, rotated rx 180 ry 0 rz 90 deg; joints [4.101, -66.36, 104.817, -11.657, 12.872, 14.561]
  MoveL 595 to (-783.4, 550, 50) mm, rotated rx -180 ry 0 rz 90 deg; joints [4.224, -68.338, 107.76, -12.936, 11.949, 15.95]
  MoveL 596 to (-783.4, 550, -0.5) mm, rotated rx -180 ry 0 rz 90 deg; joints [4.224, -66.527, 108.317, -16.042, 9.656, 19.111]
  MoveL 597 to (-783.4, 550, 50) mm, rotated rx -180 ry 0 rz 90 deg; joints [4.224, -68.338, 107.76, -12.936, 11.949, 15.95]
  MoveL 598 to (-783.4, 600, 50) mm, rotated rx -180 ry 0 rz 90 deg; joints [4.354, -70.323, 110.645, -14.37, 11.098, 17.498]
  MoveL 599 to (-783.4, 600, -0.5) mm, rotated rx 180 ry 0 rz 90 deg; joints [4.354, -68.443, 111.213, -18.309, 8.747, 21.496]
  MoveL 600 to (-783.4, 600, 50) mm, rotated rx -180 ry 0 rz 90 deg; joints [4.354, -70.323, 110.645, -14.37, 11.098, 17.498]
  MoveL 601 to (-783.4, 650, 50) mm, rotated rx -180 ry 0 rz 90 deg; joints [4.492, -72.321, 113.478, -15.968, 10.32, 19.216]
  MoveL 602 to (-783.4, 650, -0.5) mm, rotated rx 180 ry 0 rz 90 deg; joints [4.492, -70.368, 114.059, -20.975, 7.914, 24.285]
  MoveL 603 to (-783.4, 650, 50) mm, rotated rx -180 ry 0 rz 90 deg; joints [4.492, -72.321, 113.478, -15.968, 10.32, 19.216]
  MoveL 604 to (-783.4, 700, 50) mm, rotated rx 180 ry 0 rz 90 deg; joints [4.639, -74.34, 116.261, -17.731, 9.62, 21.104]
  MoveL 605 to (-783.4, 700, -0.5) mm, rotated rx -180 ry 0 rz 90 deg; joints [4.639, -72.308, 116.857, -24.092, 7.162, 27.534]
  MoveL 606 to (-783.4, 700, 50) mm, rotated rx 180 ry 0 rz 90 deg; joints [4.639, -74.34, 116.261, -17.731, 9.62, 21.104]
  MoveL 607 to (-783.4, 750, 50) mm, rotated rx 180 ry 0 rz 90 deg; joints [4.796, -76.386, 118.998, -19.646, 9.003, 23.153]
  MoveL 608 to (-783.4, 750, -0.5) mm, rotated rx 180 ry 0 rz 90 deg; joints [4.796, -74.271, 119.61, -27.701, 6.499, 31.279]
  MoveL 609 to (-783.4, 750, 50) mm, rotated rx 180 ry 0 rz 90 deg; joints [4.796, -76.386, 118.998, -19.646, 9.003, 23.153]
  MoveL 610 to (-783.4, 800, 50) mm, rotated rx 180 ry 0 rz 90 deg; joints [4.963, -78.467, 121.691, -21.687, 8.473, 25.333]
  MoveL 611 to (-783.4, 800, -0.5) mm, rotated rx 180 ry 0 rz 90 deg; joints [4.963, -76.263, 122.322, -31.799, 5.931, 35.522]
  MoveL 612 to (-783.4, 800, 50) mm, rotated rx 180 ry 0 rz 90 deg; joints [4.963, -78.467, 121.691, -21.687, 8.473, 25.333]
  MoveL 613 to (-783.4, 850, 50) mm, rotated rx 180 ry 0 rz 90 deg; joints [5.144, -80.592, 124.343, -23.798, 8.037, 27.591]
  MoveL 614 to (-783.4, 850, -0.5) mm, rotated rx -180 ry 0 rz 90 deg; joints [5.144, -78.292, 124.995, -36.314, 5.467, 40.191]
  MoveL 615 to (-783.4, 850, 50) mm, rotated rx 180 ry 0 rz 90 deg; joints [5.144, -80.592, 124.343, -23.798, 8.037, 27.591]
  MoveL 616 to (-783.4, 900, 50) mm, rotated rx -180 ry 0 rz 90 deg; joints [5.337, -82.77, 126.955, -25.898, 7.702, 29.847]
  MoveL 617 to (-783.4, 900, -0.5) mm, rotated rx 180 ry 0 rz 90 deg; joints [5.337, -80.368, 127.631, -41.071, 5.112, 45.111]
  MoveL 618 to (-783.4, 900, 50) mm, rotated rx -180 ry 0 rz 90 deg; joints [5.337, -82.77, 126.955, -25.898, 7.702, 29.847]
  MoveL 619 to (-783.4, 950, 50) mm, rotated rx 180 ry 0 rz 90 deg; joints [5.546, -85.013, 129.529, -27.874, 7.474, 31.988]
  MoveL 620 to (-783.4, 950, -0.5) mm, rotated rx 180 ry 0 rz 90 deg; joints [5.546, -82.5, 130.232, -45.776, 4.868, 49.988]
  MoveL 621 to (-783.4, 950, 50) mm, rotated rx 180 ry 0 rz 90 deg; joints [5.546, -85.013, 129.529, -27.874, 7.474, 31.988]
  MoveL 622 to (-783.4, 1000, 50) mm, rotated rx 180 ry 0 rz 90 deg; joints [5.771, -87.334, 132.066, -29.594, 7.362, 33.882]
  MoveL 623 to (-783.4, 1000, -0.5) mm, rotated rx 180 ry 0 rz 90 deg; joints [5.771, -84.702, 132.798, -50.037, 4.736, 54.432]
  MoveL 624 to (-783.4, 1000, 50) mm, rotated rx 180 ry 0 rz 90 deg; joints [5.771, -87.334, 132.066, -29.594, 7.362, 33.882]
  MoveL 625 to (-783.4, 1050, 50) mm, rotated rx 180 ry 0 rz 90 deg; joints [6.016, -89.748, 134.565, -30.916, 7.376, 35.389]
  MoveL 626 to (-783.4, 1050, -0.5) mm, rotated rx 180 ry 0 rz 90 deg; joints [6.016, -86.988, 135.331, -53.43, 4.711, 58.02]
  MoveL 627 to (-783.4, 1050, 50) mm, rotated rx 180 ry 0 rz 90 deg; joints [6.016, -89.748, 134.565, -30.916, 7.376, 35.389]
  MoveL 628 to (-783.4, 1100, 50) mm, rotated rx -180 ry 0 rz 90 deg; joints [6.282, -92.272, 137.028, -31.716, 7.527, 36.385]
  MoveL 629 to (-783.4, 1100, -0.5) mm, rotated rx 180 ry 0 rz 90 deg; joints [6.282, -89.374, 137.832, -55.581, 4.789, 60.378]
  MoveL 630 to (-783.4, 1100, 50) mm, rotated rx -180 ry 0 rz 90 deg; joints [6.282, -92.272, 137.028, -31.716, 7.527, 36.385]
  MoveL 631 to (-783.4, 1150, 50) mm, rotated rx 180 ry 0 rz 90 deg; joints [6.573, -94.93, 139.452, -31.906, 7.834, 36.783]
  MoveL 632 to (-783.4, 1150, -0.5) mm, rotated rx 180 ry 0 rz 90 deg; joints [6.573, -91.883, 140.3, -56.229, 4.972, 61.246]
  MoveL 633 to (-783.4, 1150, 50) mm, rotated rx 180 ry 0 rz 90 deg; joints [6.573, -94.93, 139.452, -31.906, 7.834, 36.783]
  MoveL 634 to (-783.4, 1200, 50) mm, rotated rx -180 ry 0 rz 90 deg; joints [6.892, -97.746, 141.838, -31.458, 8.32, 36.555]
  MoveL 635 to (-783.4, 1200, -0.5) mm, rotated rx 180 ry 0 rz 90 deg; joints [6.892, -94.541, 142.734, -55.266, 5.273, 60.518]
  MoveL 636 to (-783.4, 1200, 50) mm, rotated rx -180 ry 0 rz 90 deg; joints [6.892, -97.746, 141.838, -31.458, 8.32, 36.555]
  MoveL 637 to (-783.4, 1250, 50) mm, rotated rx 180 ry 0 rz 90 deg; joints [7.243, -100.753, 144.182, -30.407, 9.019, 35.738]
  MoveL 638 to (-783.4, 1250, -0.5) mm, rotated rx -180 ry 0 rz 90 deg; joints [7.243, -97.379, 145.134, -52.754, 5.721, 58.257]
  MoveL 639 to (-783.4, 1250, 50) mm, rotated rx 180 ry 0 rz 90 deg; joints [7.243, -100.753, 144.182, -30.407, 9.019, 35.738]
  MoveL 640 to (-681, 1150, 50) mm, rotated rx -180 ry 0 rz 90 deg; joints [1.123, -95.31, 139.785, -6.193, 6.568, 7.026]
  MoveL 641 to (-681, 1150, -0.5) mm, rotated rx 180 ry 0 rz 90 deg; joints [1.123, -92.242, 140.639, -15.17, 2.703, 16.027]
  MoveL 642 to (-681, 1150, 50) mm, rotated rx -180 ry 0 rz 90 deg; joints [1.123, -95.31, 139.785, -6.193, 6.568, 7.026]
  MoveL 643 to (-719.2, 1150, 50) mm, rotated rx 180 ry 0 rz 90 deg; joints [3.164, -95.23, 139.716, -16.929, 6.851, 19.275]
  MoveL 644 to (-719.2, 1150, -0.5) mm, rotated rx 180 ry 0 rz 90 deg; joints [3.164, -92.167, 140.568, -37.022, 3.307, 39.436]
  MoveL 645 to (-719.2, 1150, 50) mm, rotated rx 180 ry 0 rz 90 deg; joints [3.164, -95.23, 139.716, -16.929, 6.851, 19.275]
  MoveL 646 to (-757.4, 1150, 50) mm, rotated rx 180 ry 0 rz 90 deg; joints [5.197, -95.077, 139.581, -26.38, 7.371, 30.234]
  MoveL 647 to (-757.4, 1150, -0.5) mm, rotated rx -180 ry 0 rz 90 deg; joints [5.197, -92.022, 140.431, -50.411, 4.242, 54.377]
  MoveL 648 to (-757.4, 1150, 50) mm, rotated rx 180 ry 0 rz 90 deg; joints [5.197, -95.077, 139.581, -26.38, 7.371, 30.234]
  MoveL 649 to (-890, 50, 50) mm, rotated rx -180 ry 0 rz 90 deg; joints [6.048, -47.461, 73.968, -9.053, 24.923, 12.929]
  MoveL 650 to (-890, 50, -0.5) mm, rotated rx 180 ry 0 rz 90 deg; joints [6.048, -46.191, 74.507, -9.715, 23.137, 13.653]
  MoveL 651 to (-890, 50, 50) mm, rotated rx -180 ry 0 rz 90 deg; joints [6.048, -47.461, 73.968, -9.053, 24.923, 12.929]
  MoveL 652 to (-890, 100, 50) mm, rotated rx -180 ry 0 rz 90 deg; joints [6.189, -49.672, 77.785, -9.853, 23.359, 13.877]
  MoveL 653 to (-890, 100, -0.5) mm, rotated rx 180 ry 0 rz 90 deg; joints [6.189, -48.356, 78.316, -10.649, 21.541, 14.738]
  MoveL 654 to (-890, 100, 50) mm, rotated rx -180 ry 0 rz 90 deg; joints [6.189, -49.672, 77.785, -9.853, 23.359, 13.877]
  MoveL 655 to (-890, 150, 50) mm, rotated rx 180 ry 0 rz 90 deg; joints [6.337, -51.821, 81.452, -10.739, 21.889, 14.914]
  MoveL 656 to (-890, 150, -0.5) mm, rotated rx 180 ry 0 rz 90 deg; joints [6.337, -50.46, 81.978, -11.697, 20.037, 15.94]
  MoveL 657 to (-890, 150, 50) mm, rotated rx 180 ry 0 rz 90 deg; joints [6.337, -51.821, 81.452, -10.739, 21.889, 14.914]
  MoveL 658 to (-890, 200, 50) mm, rotated rx 180 ry 0 rz 90 deg; joints [6.493, -53.921, 84.988, -11.721, 20.507, 16.051]
  MoveL 659 to (-890, 200, -0.5) mm, rotated rx -180 ry 0 rz 90 deg; joints [6.493, -52.513, 85.512, -12.879, 18.619, 17.281]
  MoveL 660 to (-890, 200, 50) mm, rotated rx 180 ry 0 rz 90 deg; joints [6.493, -53.921, 84.988, -11.721, 20.507, 16.051]
  MoveL 661 to (-890, 250, 50) mm, rotated rx 180 ry 0 rz 90 deg; joints [6.656, -55.981, 88.409, -12.812, 19.206, 17.302]
  MoveL 662 to (-890, 250, -0.5) mm, rotated rx -180 ry 0 rz 90 deg; joints [6.656, -54.524, 88.932, -14.216, 17.28, 18.78]
  MoveL 663 to (-890, 250, 50) mm, rotated rx 180 ry 0 rz 90 deg; joints [6.656, -55.981, 88.409, -12.812, 19.206, 17.302]
  MoveL 664 to (-890, 300, 50) mm, rotated rx 180 ry 0 rz 90 deg; joints [6.828, -58.008, 91.728, -14.025, 17.983, 18.681]
  MoveL 665 to (-890, 300, -0.5) mm, rotated rx 180 ry 0 rz 90 deg; joints [6.828, -56.501, 92.252, -15.731, 16.019, 20.465]
  MoveL 666 to (-890, 300, 50) mm, rotated rx 180 ry 0 rz 90 deg; joints [6.828, -58.008, 91.728, -14.025, 17.983, 18.681]
  MoveL 667 to (-890, 350, 50) mm, rotated rx 180 ry 0 rz 90 deg; joints [7.008, -60.01, 94.954, -15.374, 16.836, 20.202]
  MoveL 668 to (-890, 350, -0.5) mm, rotated rx -180 ry 0 rz 90 deg; joints [7.008, -58.451, 95.482, -17.454, 14.833, 22.363]
  MoveL 669 to (-890, 350, 50) mm, rotated rx 180 ry 0 rz 90 deg; joints [7.008, -60.01, 94.954, -15.374, 16.836, 20.202]
  MoveL 670 to (-890, 400, 50) mm, rotated rx 180 ry 0 rz 90 deg; joints [7.199, -61.993, 98.098, -16.875, 15.764, 21.881]
  MoveL 671 to (-890, 400, -0.5) mm, rotated rx 180 ry 0 rz 90 deg; joints [7.199, -60.379, 98.63, -19.416, 13.724, 24.508]
  MoveL 672 to (-890, 400, 50) mm, rotated rx 180 ry 0 rz 90 deg; joints [7.199, -61.993, 98.098, -16.875, 15.764, 21.881]
  MoveL 673 to (-890, 450, 50) mm, rotated rx -180 ry 0 rz 90 deg; joints [7.4, -63.964, 101.167, -18.542, 14.767, 23.733]
  MoveL 674 to (-890, 450, -0.5) mm, rotated rx 180 ry 0 rz 90 deg; joints [7.4, -62.293, 101.705, -21.65, 12.691, 26.932]
  MoveL 675 to (-890, 450, 50) mm, rotated rx -180 ry 0 rz 90 deg; joints [7.4, -63.964, 101.167, -18.542, 14.767, 23.733]
  MoveL 676 to (-890, 500, 50) mm, rotated rx -180 ry 0 rz 90 deg; joints [7.612, -65.929, 104.167, -20.386, 13.847, 25.77]
  MoveL 677 to (-890, 500, -0.5) mm, rotated rx -180 ry 0 rz 90 deg; joints [7.612, -64.197, 104.713, -24.192, 11.738, 29.672]
  MoveL 678 to (-890, 500, 50) mm, rotated rx -180 ry 0 rz 90 deg; joints [7.612, -65.929, 104.167, -20.386, 13.847, 25.77]
  MoveL 679 to (-890, 550, 50) mm, rotated rx 180 ry 0 rz 90 deg; joints [7.837, -67.893, 107.103, -22.417, 13.005, 28.003]
  MoveL 680 to (-890, 550, -0.5) mm, rotated rx -180 ry 0 rz 90 deg; joints [7.837, -66.097, 107.658, -27.074, 10.868, 32.761]
  MoveL 681 to (-890, 550, 50) mm, rotated rx 180 ry 0 rz 90 deg; joints [7.837, -67.893, 107.103, -22.417, 13.005, 28.003]
  MoveL 682 to (-890, 600, 50) mm, rotated rx -180 ry 0 rz 90 deg; joints [8.076, -69.862, 109.982, -24.637, 12.245, 30.434]
  MoveL 683 to (-890, 600, -0.5) mm, rotated rx 180 ry 0 rz 90 deg; joints [8.076, -67.998, 110.547, -30.318, 10.087, 36.224]
  MoveL 684 to (-890, 600, 50) mm, rotated rx -180 ry 0 rz 90 deg; joints [8.076, -69.862, 109.982, -24.637, 12.245, 30.434]
  MoveL 685 to (-890, 650, 50) mm, rotated rx 180 ry 0 rz 90 deg; joints [8.33, -71.842, 112.806, -27.038, 11.569, 33.056]
  MoveL 686 to (-890, 650, -0.5) mm, rotated rx 180 ry 0 rz 90 deg; joints [8.33, -69.907, 113.383, -33.934, 9.399, 40.068]
  MoveL 687 to (-890, 650, 50) mm, rotated rx 180 ry 0 rz 90 deg; joints [8.33, -71.842, 112.806, -27.038, 11.569, 33.056]
  MoveL 688 to (-890, 700, 50) mm, rotated rx 180 ry 0 rz 90 deg; joints [8.599, -73.84, 115.579, -29.6, 10.982, 35.85]
  MoveL 689 to (-890, 700, -0.5) mm, rotated rx 180 ry 0 rz 90 deg; joints [8.599, -71.828, 116.171, -37.9, 8.812, 44.274]
  MoveL 690 to (-890, 700, 50) mm, rotated rx 180 ry 0 rz 90 deg; joints [8.599, -73.84, 115.579, -29.6, 10.982, 35.85]
  MoveL 691 to (-890, 750, 50) mm, rotated rx -180 ry 0 rz 90 deg; joints [8.887, -75.861, 118.304, -32.283, 10.488, 38.777]
  MoveL 692 to (-890, 750, -0.5) mm, rotated rx 180 ry 0 rz 90 deg; joints [8.887, -73.768, 118.912, -42.157, 8.329, 48.783]
  MoveL 693 to (-890, 750, 50) mm, rotated rx -180 ry 0 rz 90 deg; joints [8.887, -75.861, 118.304, -32.283, 10.488, 38.777]
  MoveL 694 to (-890, 800, 50) mm, rotated rx -180 ry 0 rz 90 deg; joints [9.195, -77.914, 120.985, -35.025, 10.091, 41.776]
  MoveL 695 to (-890, 800, -0.5) mm, rotated rx 180 ry 0 rz 90 deg; joints [9.195, -75.734, 121.611, -46.596, 7.956, 53.489]
  MoveL 696 to (-890, 800, 50) mm, rotated rx -180 ry 0 rz 90 deg; joints [9.195, -77.914, 120.985, -35.025, 10.091, 41.776]
  MoveL 697 to (-890, 850, 50) mm, rotated rx 180 ry 0 rz 90 deg; joints [9.524, -80.006, 123.622, -37.745, 9.794, 44.768]
  MoveL 698 to (-890, 850, -0.5) mm, rotated rx 180 ry 0 rz 90 deg; joints [9.524, -77.733, 124.268, -51.059, 7.694, 58.234]
  MoveL 699 to (-890, 850, 50) mm, rotated rx 180 ry 0 rz 90 deg; joints [9.524, -80.006, 123.622, -37.745, 9.794, 44.768]
  MoveL 700 to (-890, 900, 50) mm, rotated rx 180 ry 0 rz 90 deg; joints [9.877, -82.146, 126.218, -40.341, 9.6, 47.649]
  MoveL 701 to (-890, 900, -0.5) mm, rotated rx 180 ry 0 rz 90 deg; joints [9.877, -79.774, 126.887, -55.35, 7.541, 62.823]
  MoveL 702 to (-890, 900, 50) mm, rotated rx 180 ry 0 rz 90 deg; joints [9.877, -82.146, 126.218, -40.341, 9.6, 47.649]
  MoveL 703 to (-890, 950, 50) mm, rotated rx 180 ry 0 rz 90 deg; joints [10.258, -84.345, 128.775, -42.697, 9.513, 50.307]
  MoveL 704 to (-890, 950, -0.5) mm, rotated rx 180 ry 0 rz 90 deg; joints [10.258, -81.865, 129.469, -59.253, 7.493, 67.042]
  MoveL 705 to (-890, 950, 50) mm, rotated rx 180 ry 0 rz 90 deg; joints [10.258, -84.345, 128.775, -42.697, 9.513, 50.307]
  MoveL 706 to (-890, 1000, 50) mm, rotated rx -180 ry 0 rz 90 deg; joints [10.669, -86.613, 131.292, -44.694, 9.535, 52.625]
  MoveL 707 to (-890, 1000, -0.5) mm, rotated rx 180 ry 0 rz 90 deg; joints [10.669, -84.019, 132.015, -62.563, 7.543, 70.688]
  MoveL 708 to (-890, 1000, 50) mm, rotated rx -180 ry 0 rz 90 deg; joints [10.669, -86.613, 131.292, -44.694, 9.535, 52.625]
  MoveL 709 to (-890, 1050, 50) mm, rotated rx 180 ry 0 rz 90 deg; joints [11.113, -88.965, 133.77, -46.224, 9.671, 54.494]
  MoveL 710 to (-890, 1050, -0.5) mm, rotated rx -180 ry 0 rz 90 deg; joints [11.113, -86.247, 134.525, -65.106, 7.685, 73.587]
  MoveL 711 to (-890, 1050, 50) mm, rotated rx 180 ry 0 rz 90 deg; joints [11.113, -88.965, 133.77, -46.224, 9.671, 54.494]
  MoveL 712 to (-890, 1100, 50) mm, rotated rx 180 ry 0 rz 90 deg; joints [11.596, -91.416, 136.21, -47.195, 9.928, 55.825]
  MoveL 713 to (-890, 1100, -0.5) mm, rotated rx -180 ry 0 rz 90 deg; joints [11.596, -88.566, 137.001, -66.749, 7.913, 75.61]
  MoveL 714 to (-890, 1100, 50) mm, rotated rx 180 ry 0 rz 90 deg; joints [11.596, -91.416, 136.21, -47.195, 9.928, 55.825]
  MoveL 715 to (-890, 1150, 50) mm, rotated rx -180 ry 0 rz 90 deg; joints [12.121, -93.986, 138.611, -47.547, 10.317, 56.557]
  MoveL 716 to (-890, 1150, -0.5) mm, rotated rx 180 ry 0 rz 90 deg; joints [12.121, -90.992, 139.442, -67.405, 8.229, 76.67]
  MoveL 717 to (-890, 1150, 50) mm, rotated rx -180 ry 0 rz 90 deg; joints [12.121, -93.986, 138.611, -47.547, 10.317, 56.557]
  MoveL 718 to (-890, 1200, 50) mm, rotated rx 180 ry 0 rz 90 deg; joints [12.696, -96.696, 140.97, -47.251, 10.857, 56.665]
  MoveL 719 to (-890, 1200, -0.5) mm, rotated rx -180 ry 0 rz 90 deg; joints [12.696, -93.55, 141.848, -67.027, 8.64, 76.722]
  MoveL 720 to (-890, 1200, 50) mm, rotated rx 180 ry 0 rz 90 deg; joints [12.696, -96.696, 140.97, -47.251, 10.857, 56.665]
  MoveL 721 to (-890, 1250, 50) mm, rotated rx -180 ry 0 rz 90 deg; joints [13.327, -99.573, 143.287, -46.319, 11.571, 56.162]
  MoveL 722 to (-890, 1250, -0.5) mm, rotated rx -180 ry 0 rz 90 deg; joints [13.327, -96.265, 144.216, -65.611, 9.165, 75.764]
  MoveL 723 to (-890, 1250, 50) mm, rotated rx -180 ry 0 rz 90 deg; joints [13.327, -99.573, 143.287, -46.319, 11.571, 56.162]
  MoveL 724 to (-890, 1300, 50) mm, rotated rx 180 ry 0 rz 90 deg; joints [14.023, -102.65, 145.557, -44.802, 12.498, 55.099]
  MoveL 725 to (-890, 1300, -0.5) mm, rotated rx -180 ry 0 rz 90 deg; joints [14.023, -99.171, 146.545, -63.197, 9.837, 73.839]
  MoveL 726 to (-890, 1300, 50) mm, rotated rx 180 ry 0 rz 90 deg; joints [14.023, -102.65, 145.557, -44.802, 12.498, 55.099]
  MoveL 727 to (-890, 1350, 50) mm, rotated rx 180 ry 0 rz 90 deg; joints [14.794, -105.966, 147.776, -42.786, 13.684, 53.562]
  MoveL 728 to (-890, 1350, -0.5) mm, rotated rx 180 ry 0 rz 90 deg; joints [14.794, -102.309, 148.832, -59.883, 10.706, 71.043]
  MoveL 729 to (-890, 1350, 50) mm, rotated rx 180 ry 0 rz 90 deg; joints [14.794, -105.966, 147.776, -42.786, 13.684, 53.562]
  MoveL 730 to (-890, 1400, 50) mm, rotated rx 180 ry 0 rz 90 deg; joints [15.652, -109.569, 149.938, -40.386, 15.191, 51.667]
  MoveL 731 to (-890, 1400, -0.5) mm, rotated rx -180 ry 0 rz 90 deg; joints [15.652, -105.733, 151.071, -55.828, 11.842, 67.536]
  MoveL 732 to (-890, 1400, 50) mm, rotated rx 180 ry 0 rz 90 deg; joints [15.652, -109.569, 149.938, -40.386, 15.191, 51.667]
  MoveL 733 to (-890, 1450, 50) mm, rotated rx 180 ry 0 rz 90 deg; joints [16.612, -113.516, 152.035, -37.737, 17.096, 49.546]
  MoveL 734 to (-890, 1450, -0.5) mm, rotated rx 180 ry 0 rz 90 deg; joints [16.612, -109.508, 153.256, -51.25, 13.338, 63.537]
  MoveL 735 to (-890, 1450, 50) mm, rotated rx 180 ry 0 rz 90 deg; joints [16.612, -113.516, 152.035, -37.737, 17.096, 49.546]
  MoveL 736 to (-960, 50, 50) mm, rotated rx 180 ry 0 rz 90 deg; joints [7.868, -47.077, 73.301, -11.546, 25.493, 16.578]
  MoveL 737 to (-960, 50, -0.5) mm, rotated rx 180 ry 0 rz 90 deg; joints [7.868, -45.814, 73.841, -12.362, 23.729, 17.475]
  MoveL 738 to (-960, 50, 50) mm, rotated rx 180 ry 0 rz 90 deg; joints [7.868, -47.077, 73.301, -11.546, 25.493, 16.578]
  MoveL 739 to (-960, 100, 50) mm, rotated rx 180 ry 0 rz 90 deg; joints [8.051, -49.291, 77.13, -12.542, 23.947, 17.765]
  MoveL 740 to (-960, 100, -0.5) mm, rotated rx 180 ry 0 rz 90 deg; joints [8.051, -47.983, 77.663, -13.517, 22.154, 18.825]
  MoveL 741 to (-960, 100, 50) mm, rotated rx 180 ry 0 rz 90 deg; joints [8.051, -49.291, 77.13, -12.542, 23.947, 17.765]
  MoveL 742 to (-960, 150, 50) mm, rotated rx 180 ry 0 rz 90 deg; joints [8.243, -51.441, 80.806, -13.637, 22.499, 19.057]
  MoveL 743 to (-960, 150, -0.5) mm, rotated rx 180 ry 0 rz 90 deg; joints [8.243, -50.088, 81.334, -14.805, 20.676, 20.313]
  MoveL 744 to (-960, 150, 50) mm, rotated rx 180 ry 0 rz 90 deg; joints [8.243, -51.441, 80.806, -13.637, 22.499, 19.057]
  MoveL 745 to (-960, 200, 50) mm, rotated rx 180 ry 0 rz 90 deg; joints [8.444, -53.54, 84.349, -14.845, 21.142, 20.467]
  MoveL 746 to (-960, 200, -0.5) mm, rotated rx 180 ry 0 rz 90 deg; joints [8.444, -52.14, 84.874, -16.246, 19.288, 21.959]
  MoveL 747 to (-960, 200, 50) mm, rotated rx 180 ry 0 rz 90 deg; joints [8.444, -53.54, 84.349, -14.845, 21.142, 20.467]
  MoveL 748 to (-960, 250, 50) mm, rotated rx -180 ry 0 rz 90 deg; joints [8.655, -55.597, 87.775, -16.177, 19.871, 22.006]
  MoveL 749 to (-960, 250, -0.5) mm, rotated rx -180 ry 0 rz 90 deg; joints [8.655, -54.149, 88.298, -17.86, 17.986, 23.785]
  MoveL 750 to (-960, 250, 50) mm, rotated rx -180 ry 0 rz 90 deg; joints [8.655, -55.597, 87.775, -16.177, 19.871, 22.006]
  MoveL 751 to (-960, 300, 50) mm, rotated rx -180 ry 0 rz 90 deg; joints [8.877, -57.62, 91.096, -17.647, 18.683, 23.69]
  MoveL 752 to (-960, 300, -0.5) mm, rotated rx -180 ry 0 rz 90 deg; joints [8.877, -56.122, 91.62, -19.67, 16.768, 25.815]
  MoveL 753 to (-960, 300, 50) mm, rotated rx -180 ry 0 rz 90 deg; joints [8.877, -57.62, 91.096, -17.647, 18.683, 23.69]
  MoveL 754 to (-960, 350, 50) mm, rotated rx -180 ry 0 rz 90 deg; joints [9.11, -59.616, 94.323, -19.266, 17.576, 25.532]
  MoveL 755 to (-960, 350, -0.5) mm, rotated rx 180 ry 0 rz 90 deg; joints [9.11, -58.067, 94.85, -21.703, 15.631, 28.074]
  MoveL 756 to (-960, 350, 50) mm, rotated rx -180 ry 0 rz 90 deg; joints [9.11, -59.616, 94.323, -19.266, 17.576, 25.532]
  MoveL 757 to (-960, 400, 50) mm, rotated rx 180 ry 0 rz 90 deg; joints [9.356, -61.592, 97.466, -21.048, 16.55, 27.544]
  MoveL 758 to (-960, 400, -0.5) mm, rotated rx -180 ry 0 rz 90 deg; joints [9.356, -59.989, 97.997, -23.982, 14.578, 30.59]
  MoveL 759 to (-960, 400, 50) mm, rotated rx 180 ry 0 rz 90 deg; joints [9.356, -61.592, 97.466, -21.048, 16.55, 27.544]
  MoveL 760 to (-960, 450, 50) mm, rotated rx -180 ry 0 rz 90 deg; joints [9.615, -63.553, 100.532, -23.002, 15.604, 29.738]
  MoveL 761 to (-960, 450, -0.5) mm, rotated rx 180 ry 0 rz 90 deg; joints [9.615, -61.894, 101.069, -26.533, 13.609, 33.387]
  MoveL 762 to (-960, 450, 50) mm, rotated rx -180 ry 0 rz 90 deg; joints [9.615, -63.553, 100.532, -23.002, 15.604, 29.738]
  MoveL 763 to (-960, 500, 50) mm, rotated rx -180 ry 0 rz 90 deg; joints [9.889, -65.507, 103.528, -25.134, 14.741, 32.12]
  MoveL 764 to (-960, 500, -0.5) mm, rotated rx 180 ry 0 rz 90 deg; joints [9.889, -63.788, 104.072, -29.376, 12.728, 36.486]
  MoveL 765 to (-960, 500, 50) mm, rotated rx -180 ry 0 rz 90 deg; joints [9.889, -65.507, 103.528, -25.134, 14.741, 32.12]
  MoveL 766 to (-960, 550, 50) mm, rotated rx 180 ry 0 rz 90 deg; joints [10.179, -67.458, 106.459, -27.445, 13.963, 34.692]
  MoveL 767 to (-960, 550, -0.5) mm, rotated rx -180 ry 0 rz 90 deg; joints [10.179, -65.676, 107.011, -32.521, 11.939, 39.898]
  MoveL 768 to (-960, 550, 50) mm, rotated rx 180 ry 0 rz 90 deg; joints [10.179, -67.458, 106.459, -27.445, 13.963, 34.692]
  MoveL 769 to (-960, 600, 50) mm, rotated rx 180 ry 0 rz 90 deg; joints [10.486, -69.412, 109.33, -29.927, 13.272, 37.446]
  MoveL 770 to (-960, 600, -0.5) mm, rotated rx -180 ry 0 rz 90 deg; joints [10.486, -67.564, 109.893, -35.965, 11.246, 43.623]
  MoveL 771 to (-960, 600, 50) mm, rotated rx 180 ry 0 rz 90 deg; joints [10.486, -69.412, 109.33, -29.927, 13.272, 37.446]
  MoveL 772 to (-960, 650, 50) mm, rotated rx -180 ry 0 rz 90 deg; joints [10.812, -71.375, 112.146, -32.559, 12.671, 40.363]
  MoveL 773 to (-960, 650, -0.5) mm, rotated rx 180 ry 0 rz 90 deg; joints [10.812, -69.457, 112.721, -39.685, 10.653, 47.638]
  MoveL 774 to (-960, 650, 50) mm, rotated rx -180 ry 0 rz 90 deg; joints [10.812, -71.375, 112.146, -32.559, 12.671, 40.363]
  MoveL 775 to (-960, 700, 50) mm, rotated rx 180 ry 0 rz 90 deg; joints [11.158, -73.353, 114.909, -35.307, 12.164, 43.411]
  MoveL 776 to (-960, 700, -0.5) mm, rotated rx -180 ry 0 rz 90 deg; joints [11.158, -71.36, 115.498, -43.629, 10.166, 51.891]
  MoveL 777 to (-960, 700, 50) mm, rotated rx 180 ry 0 rz 90 deg; joints [11.158, -73.353, 114.909, -35.307, 12.164, 43.411]
  MoveL 778 to (-960, 750, 50) mm, rotated rx -180 ry 0 rz 90 deg; joints [11.528, -75.351, 117.624, -38.122, 11.755, 46.541]
  MoveL 779 to (-960, 750, -0.5) mm, rotated rx 180 ry 0 rz 90 deg; joints [11.528, -73.279, 118.228, -47.714, 9.788, 56.302]
  MoveL 780 to (-960, 750, 50) mm, rotated rx -180 ry 0 rz 90 deg; joints [11.528, -75.351, 117.624, -38.122, 11.755, 46.541]
  MoveL 781 to (-960, 800, 50) mm, rotated rx 180 ry 0 rz 90 deg; joints [11.922, -77.377, 120.292, -40.937, 11.444, 49.686]
